LIN {X 0,Y 368.293,Z 314.692,A -85,B 0,C 180,E1 -12573.966,E2 -12573.966} C_VEL
LIN {X 0,Y 368.178,Z 320.417,A -85,B 0,C 180,E1 -12577.556,E2 -12577.556} C_VEL
LIN {X 0,Y 368.144,Z 324.235,A -85,B 0,C 180,E1 -12579.902,E2 -12579.902} C_VEL
LIN {X 0,Y 368.132,Z 327.336,A -85,B 0,C 180,E1 -12581.747,E2 -12581.747} C_VEL
LIN {X 0,Y 370.901,Z 341.005,A -85,B 0,C 180,E1 -12582.407,E2 -12582.407} C_VEL
LIN {X 0,Y 372.726,Z 351.323,A -85,B 0,C 180,E1 -12583.051,E2 -12583.051} C_VEL
LIN {X 0,Y 372.036,Z 364.185,A -85,B 0,C 180,E1 -12583.962,E2 -12583.962} C_VEL
LIN {X 0,Y 371.306,Z 375.959,A -85,B 0,C 180,E1 -12585.036,E2 -12585.036} C_VEL
LIN {X 0,Y 370.622,Z 386.995,A -85,B 0,C 180,E1 -12586.288,E2 -12586.288} C_VEL
LIN {X 0,Y 369.859,Z 396.767,A -85,B 0,C 180,E1 -12587.656,E2 -12587.656} C_VEL
LIN {X 0,Y 369.188,Z 406.325,A -85,B 0,C 180,E1 -12589.304,E2 -12589.304} C_VEL
LIN {X 0,Y 368.622,Z 413.953,A -85,B 0,C 180,E1 -12590.95,E2 -12590.95} C_VEL
LIN {X 0,Y 368.197,Z 420.432,A -85,B 0,C 180,E1 -12592.693,E2 -12592.693} C_VEL
LIN {X 0,Y 367.947,Z 425.635,A -85,B 0,C 180,E1 -12594.52,E2 -12594.52} C_VEL
LIN {X 0,Y 367.836,Z 428.082,A -85,B 0,C 180,E1 -12595.617,E2 -12595.617} C_VEL
LIN {X 0,Y 367.823,Z 430.069,A -85,B 0,C 180,E1 -12596.714,E2 -12596.714} C_VEL
LIN {X 0,Y 367.74,Z 431.56,A -85,B 0,C 180,E1 -12597.809,E2 -12597.809} C_VEL
LIN {X 0,Y 367.646,Z 432.642,A -85,B 0,C 180,E1 -12598.905,E2 -12598.905} C_VEL
LIN {X 0,Y 367.637,Z 433.299,A -85,B 0,C 180,E1 -12600,E2 -12600} C_VEL
LIN {X 0,Y 367.683,Z 433.487,A -85,B 0,C 180,E1 -12601.095,E2 -12601.095} C_VEL
LIN {X 0,Y 367.802,Z 433.269,A -85,B 0,C 180,E1 -12602.19,E2 -12602.19} C_VEL
LIN {X 0,Y 367.965,Z 432.627,A -85,B 0,C 180,E1 -12603.285,E2 -12603.285} C_VEL
LIN {X 0,Y 368.17,Z 431.513,A -85,B 0,C 180,E1 -12604.379,E2 -12604.379} C_VEL
LIN {X 0,Y 368.307,Z 429.993,A -85,B 0,C 180,E1 -12605.475,E2 -12605.475} C_VEL
LIN {X 0,Y 368.614,Z 426.762,A -85,B 0,C 180,E1 -12607.157,E2 -12607.157} C_VEL
LIN {X 0,Y 369.223,Z 422.567,A -85,B 0,C 180,E1 -12608.759,E2 -12608.759} C_VEL
LIN {X 0,Y 370.013,Z 415.974,A -85,B 0,C 180,E1 -12610.672,E2 -12610.672} C_VEL
LIN {X 0,Y 370.794,Z 408.79,A -85,B 0,C 180,E1 -12612.312,E2 -12612.312} C_VEL
LIN {X 0,Y 371.912,Z 399.78,A -85,B 0,C 180,E1 -12613.942,E2 -12613.942} C_VEL
LIN {X 0,Y 372.991,Z 390.605,A -85,B 0,C 180,E1 -12615.295,E2 -12615.295} C_VEL
LIN {X 0,Y 374.108,Z 379.922,A -85,B 0,C 180,E1 -12616.57,E2 -12616.57} C_VEL
LIN {X 0,Y 375.291,Z 367.919,A -85,B 0,C 180,E1 -12617.717,E2 -12617.717} C_VEL
LIN {X 0,Y 376.322,Z 355.559,A -85,B 0,C 180,E1 -12618.649,E2 -12618.649} C_VEL
LIN {X 0,Y 373.799,Z 345.042,A -85,B 0,C 180,E1 -12619.536,E2 -12619.536} C_VEL
LIN {X 0,Y 369.814,Z 333.869,A -85,B 0,C 180,E1 -12620.45,E2 -12620.45} C_VEL
LIN {X 0,Y 369.281,Z 332.067,A -85,B 0,C 180,E1 -12620.593,E2 -12620.593} C_VEL
LIN {X 0,Y 369.513,Z 325.412,A -85,B 0,C 180,E1 -12624.736,E2 -12624.736} C_VEL
LIN {X 0,Y 369.884,Z 318.305,A -85,B 0,C 180,E1 -12629.07,E2 -12629.07} C_VEL
LIN {X 0,Y 370.318,Z 312.164,A -85,B 0,C 180,E1 -12632.73,E2 -12632.73} C_VEL
LIN {X 0,Y 370.032,Z 308.99,A -85,B 0,C 180,E1 -12634.736,E2 -12634.736} C_VEL
LIN {X 0,Y 368.959,Z 303.753,A -85,B 0,C 180,E1 -12638.248,E2 -12638.248} C_VEL
LIN {X 0,Y 368.903,Z 303.535,A -85,B 0,C 180,E1 -12638.953,E2 -12638.953} C_VEL
LIN {X 0,Y 368.882,Z 303.536,A -85,B 0,C 180,E1 -12642.009,E2 -12642.009} C_VEL
LIN {X 0,Y 368.969,Z 303.673,A -85,B 0,C 180,E1 -12643.414,E2 -12643.414} C_VEL
LIN {X 0,Y 370.283,Z 310.676,A -85,B 0,C 180,E1 -12646.899,E2 -12646.899} C_VEL
LIN {X 0,Y 371.896,Z 318.9,A -85,B 0,C 180,E1 -12650.788,E2 -12650.788} C_VEL
LIN {X 0,Y 372.574,Z 323.529,A -85,B 0,C 180,E1 -12652.87,E2 -12652.87} C_VEL
LIN {X 0,Y 372.208,Z 328.239,A -85,B 0,C 180,E1 -12654.861,E2 -12654.861} C_VEL
LIN {X 0,Y 371.167,Z 337.939,A -85,B 0,C 180,E1 -12658.829,E2 -12658.829} C_VEL
LIN {X 0,Y 370.182,Z 348.156,A -85,B 0,C 180,E1 -12662.893,E2 -12662.893} C_VEL
LIN {X 0,Y 369.444,Z 357.311,A -85,B 0,C 180,E1 -12666.454,E2 -12666.454} C_VEL
LIN {X 0,Y 368.798,Z 366.881,A -85,B 0,C 180,E1 -12670.121,E2 -12670.121} C_VEL
LIN {X 0,Y 370.827,Z 380.273,A -85,B 0,C 180,E1 -12670.828,E2 -12670.828} C_VEL
LIN {X 0,Y 372.37,Z 395.112,A -85,B 0,C 180,E1 -12671.806,E2 -12671.806} C_VEL
LIN {X 0,Y 373.203,Z 403.232,A -85,B 0,C 180,E1 -12672.464,E2 -12672.464} C_VEL
LIN {X 0,Y 372.141,Z 415.707,A -85,B 0,C 180,E1 -12673.544,E2 -12673.544} C_VEL
LIN {X 0,Y 371.014,Z 427.836,A -85,B 0,C 180,E1 -12674.838,E2 -12674.838} C_VEL
LIN {X 0,Y 370.307,Z 436.542,A -85,B 0,C 180,E1 -12675.996,E2 -12675.996} C_VEL
LIN {X 0,Y 369.48,Z 445.02,A -85,B 0,C 180,E1 -12677.365,E2 -12677.365} C_VEL
LIN {X 0,Y 368.646,Z 453.276,A -85,B 0,C 180,E1 -12679.01,E2 -12679.01} C_VEL
LIN {X 0,Y 368.16,Z 459.921,A -85,B 0,C 180,E1 -12680.662,E2 -12680.662} C_VEL
LIN {X 0,Y 367.808,Z 465.21,A -85,B 0,C 180,E1 -12682.313,E2 -12682.313} C_VEL
LIN {X 0,Y 367.693,Z 468.753,A -85,B 0,C 180,E1 -12683.679,E2 -12683.679} C_VEL
LIN {X 0,Y 367.561,Z 472.55,A -85,B 0,C 180,E1 -12685.614,E2 -12685.614} C_VEL
LIN {X 0,Y 367.561,Z 474.042,A -85,B 0,C 180,E1 -12686.712,E2 -12686.712} C_VEL
LIN {X 0,Y 367.596,Z 475.113,A -85,B 0,C 180,E1 -12687.809,E2 -12687.809} C_VEL
LIN {X 0,Y 367.68,Z 475.776,A -85,B 0,C 180,E1 -12688.905,E2 -12688.905} C_VEL
LIN {X 0,Y 367.674,Z 475.968,A -85,B 0,C 180,E1 -12690,E2 -12690} C_VEL
LIN {X 0,Y 367.674,Z 475.73,A -85,B 0,C 180,E1 -12691.095,E2 -12691.095} C_VEL
LIN {X 0,Y 367.623,Z 475.08,A -85,B 0,C 180,E1 -12692.191,E2 -12692.191} C_VEL
LIN {X 0,Y 367.547,Z 473.974,A -85,B 0,C 180,E1 -12693.289,E2 -12693.289} C_VEL
LIN {X 0,Y 367.571,Z 472.414,A -85,B 0,C 180,E1 -12694.386,E2 -12694.386} C_VEL
LIN {X 0,Y 367.732,Z 468.044,A -85,B 0,C 180,E1 -12696.585,E2 -12696.585} C_VEL
LIN {X 0,Y 367.909,Z 463.575,A -85,B 0,C 180,E1 -12698.237,E2 -12698.237} C_VEL
LIN {X 0,Y 368.322,Z 457.886,A -85,B 0,C 180,E1 -12699.888,E2 -12699.888} C_VEL
LIN {X 0,Y 368.894,Z 450.724,A -85,B 0,C 180,E1 -12701.539,E2 -12701.539} C_VEL
LIN {X 0,Y 369.76,Z 441.784,A -85,B 0,C 180,E1 -12703.184,E2 -12703.184} C_VEL
LIN {X 0,Y 370.829,Z 430.162,A -85,B 0,C 180,E1 -12704.931,E2 -12704.931} C_VEL
LIN {X 0,Y 372.024,Z 418.794,A -85,B 0,C 180,E1 -12706.32,E2 -12706.32} C_VEL
LIN {X 0,Y 373.408,Z 406.425,A -85,B 0,C 180,E1 -12707.526,E2 -12707.526} C_VEL
LIN {X 0,Y 373.418,Z 401.589,A -85,B 0,C 180,E1 -12707.95,E2 -12707.95} C_VEL
LIN {X 0,Y 372.561,Z 389.175,A -85,B 0,C 180,E1 -12708.946,E2 -12708.946} C_VEL
LIN {X 0,Y 371.454,Z 377.338,A -85,B 0,C 180,E1 -12709.731,E2 -12709.731} C_VEL
LIN {X 0,Y 369.366,Z 365.834,A -85,B 0,C 180,E1 -12710.417,E2 -12710.417} C_VEL
LIN {X 0,Y 368.722,Z 362.563,A -85,B 0,C 180,E1 -12710.631,E2 -12710.631} C_VEL
LIN {X 0,Y 369.355,Z 353.705,A -85,B 0,C 180,E1 -12714.03,E2 -12714.03} C_VEL
LIN {X 0,Y 370.072,Z 344.511,A -85,B 0,C 180,E1 -12717.728,E2 -12717.728} C_VEL
LIN {X 0,Y 371.079,Z 335.65,A -85,B 0,C 180,E1 -12721.54,E2 -12721.54} C_VEL
LIN {X 0,Y 372.163,Z 328.029,A -85,B 0,C 180,E1 -12725.138,E2 -12725.138} C_VEL
LIN {X 0,Y 372.658,Z 324.25,A -85,B 0,C 180,E1 -12727.121,E2 -12727.121} C_VEL
LIN {X 0,Y 372.228,Z 320.752,A -85,B 0,C 180,E1 -12729.275,E2 -12729.275} C_VEL
LIN {X 0,Y 371.416,Z 316.482,A -85,B 0,C 180,E1 -12732.441,E2 -12732.441} C_VEL
LIN {X 0,Y 370.833,Z 313.284,A -85,B 0,C 180,E1 -12735.475,E2 -12735.475} C_VEL
LIN {X 0,Y 370.417,Z 311.076,A -85,B 0,C 180,E1 -12738.389,E2 -12738.389} C_VEL
LIN {X 0,Y 370.16,Z 309.682,A -85,B 0,C 180,E1 -12741.204,E2 -12741.204} C_VEL
LIN {X 0,Y 369.927,Z 308.905,A -85,B 0,C 180,E1 -12744.779,E2 -12744.779} C_VEL
LIN {X 0,Y 369.886,Z 308.938,A -85,B 0,C 180,E1 -12747.858,E2 -12747.858} C_VEL
LIN {X 0,Y 370.009,Z 309.705,A -85,B 0,C 180,E1 -12751.65,E2 -12751.65} C_VEL
LIN {X 0,Y 370.086,Z 310.561,A -85,B 0,C 180,E1 -12754.102,E2 -12754.102} C_VEL
LIN {X 0,Y 370.024,Z 311.641,A -85,B 0,C 180,E1 -12756.493,E2 -12756.493} C_VEL
LIN {X 0,Y 369.869,Z 313.391,A -85,B 0,C 180,E1 -12759.546,E2 -12759.546} C_VEL
LIN {X 0,Y 375.177,Z 326.38,A -85,B 0,C 180,E1 -12760.749,E2 -12760.749} C_VEL
LIN {X 0,Y 377.211,Z 332.806,A -85,B 0,C 180,E1 -12761.355,E2 -12761.355} C_VEL
LIN {X 0,Y 376.25,Z 345.093,A -85,B 0,C 180,E1 -12762.295,E2 -12762.295} C_VEL
LIN {X 0,Y 375.212,Z 355.755,A -85,B 0,C 180,E1 -12763.317,E2 -12763.317} C_VEL
LIN {X 0,Y 374.169,Z 365.672,A -85,B 0,C 180,E1 -12764.475,E2 -12764.475} C_VEL
LIN {X 0,Y 373.088,Z 375.04,A -85,B 0,C 180,E1 -12765.825,E2 -12765.825} C_VEL
LIN {X 0,Y 371.984,Z 384.167,A -85,B 0,C 180,E1 -12767.451,E2 -12767.451} C_VEL
LIN {X 0,Y 370.925,Z 391.487,A -85,B 0,C 180,E1 -12769.078,E2 -12769.078} C_VEL
LIN {X 0,Y 370.181,Z 397.689,A -85,B 0,C 180,E1 -12770.838,E2 -12770.838} C_VEL
LIN {X 0,Y 369.461,Z 401.878,A -85,B 0,C 180,E1 -12772.348,E2 -12772.348} C_VEL
LIN {X 0,Y 369.123,Z 404.297,A -85,B 0,C 180,E1 -12773.44,E2 -12773.44} C_VEL
LIN {X 0,Y 368.943,Z 406.185,A -85,B 0,C 180,E1 -12774.535,E2 -12774.535} C_VEL
LIN {X 0,Y 368.636,Z 407.667,A -85,B 0,C 180,E1 -12775.626,E2 -12775.626} C_VEL
LIN {X 0,Y 368.304,Z 408.741,A -85,B 0,C 180,E1 -12776.718,E2 -12776.718} C_VEL
LIN {X 0,Y 368.069,Z 409.353,A -85,B 0,C 180,E1 -12777.811,E2 -12777.811} C_VEL
LIN {X 0,Y 367.947,Z 409.528,A -85,B 0,C 180,E1 -12778.906,E2 -12778.906} C_VEL
LIN {X 0,Y 367.9,Z 409.292,A -85,B 0,C 180,E1 -12780,E2 -12780} C_VEL
LIN {X 0,Y 367.924,Z 408.635,A -85,B 0,C 180,E1 -12781.095,E2 -12781.095} C_VEL
LIN {X 0,Y 368.046,Z 407.513,A -85,B 0,C 180,E1 -12782.189,E2 -12782.189} C_VEL
LIN {X 0,Y 368.166,Z 405.984,A -85,B 0,C 180,E1 -12783.283,E2 -12783.283} C_VEL
LIN {X 0,Y 368.432,Z 402.847,A -85,B 0,C 180,E1 -12784.924,E2 -12784.924} C_VEL
LIN {X 0,Y 368.507,Z 398.641,A -85,B 0,C 180,E1 -12786.571,E2 -12786.571} C_VEL
LIN {X 0,Y 368.886,Z 393.227,A -85,B 0,C 180,E1 -12788.215,E2 -12788.215} C_VEL
LIN {X 0,Y 369.311,Z 386.432,A -85,B 0,C 180,E1 -12789.862,E2 -12789.862} C_VEL
LIN {X 0,Y 369.939,Z 377.981,A -85,B 0,C 180,E1 -12791.506,E2 -12791.506} C_VEL
LIN {X 0,Y 370.554,Z 369.405,A -85,B 0,C 180,E1 -12792.877,E2 -12792.877} C_VEL
LIN {X 0,Y 371.324,Z 358.953,A -85,B 0,C 180,E1 -12794.244,E2 -12794.244} C_VEL
LIN {X 0,Y 372.069,Z 346.412,A -85,B 0,C 180,E1 -12795.562,E2 -12795.562} C_VEL
LIN {X 0,Y 372.687,Z 334.118,A -85,B 0,C 180,E1 -12796.572,E2 -12796.572} C_VEL
LIN {X 0,Y 373.108,Z 324.805,A -85,B 0,C 180,E1 -12797.187,E2 -12797.187} C_VEL
LIN {X 0,Y 369.814,Z 310.534,A -85,B 0,C 180,E1 -12798.046,E2 -12798.046} C_VEL
LIN {X 0,Y 368.184,Z 303.626,A -85,B 0,C 180,E1 -12798.395,E2 -12798.395} C_VEL
LIN {X 0,Y 368.516,Z 303.575,A -85,B 0,C 180,E1 -12801.245,E2 -12801.245} C_VEL
LIN {X 0,Y 368.767,Z 303.553,A -85,B 0,C 180,E1 -12803.824,E2 -12803.824} C_VEL
LIN {X 0,Y 368.916,Z 303.525,A -85,B 0,C 180,E1 -12806.443,E2 -12806.443} C_VEL
LIN {X 0,Y 368.916,Z 303.529,A -85,B 0,C 180,E1 -12809.69,E2 -12809.69} C_VEL
LIN {X 0,Y 368.901,Z 303.533,A -85,B 0,C 180,E1 -12813.044,E2 -12813.044} C_VEL
LIN {X 0,Y 368.92,Z 303.53,A -85,B 0,C 180,E1 -12816.197,E2 -12816.197} C_VEL
LIN {X 0,Y 368.905,Z 303.531,A -85,B 0,C 180,E1 -12818.953,E2 -12818.953} C_VEL
LIN {X 0,Y 368.884,Z 303.537,A -85,B 0,C 180,E1 -12822.009,E2 -12822.009} C_VEL
LIN {X 0,Y 368.883,Z 303.534,A -85,B 0,C 180,E1 -12825.176,E2 -12825.176} C_VEL
LIN {X 0,Y 368.885,Z 303.535,A -85,B 0,C 180,E1 -12828.178,E2 -12828.178} C_VEL
LIN {X 0,Y 368.91,Z 303.534,A -85,B 0,C 180,E1 -12831.36,E2 -12831.36} C_VEL
LIN {X 0,Y 368.881,Z 303.539,A -85,B 0,C 180,E1 -12833.799,E2 -12833.799} C_VEL
LIN {X 0,Y 368.808,Z 303.601,A -85,B 0,C 180,E1 -12835.96,E2 -12835.96} C_VEL
LIN {X 0,Y 368.572,Z 308.503,A -85,B 0,C 180,E1 -12839.101,E2 -12839.101} C_VEL
LIN {X 0,Y 368.516,Z 312.27,A -85,B 0,C 180,E1 -12841.525,E2 -12841.525} C_VEL
LIN {X 0,Y 368.382,Z 318.111,A -85,B 0,C 180,E1 -12845.183,E2 -12845.183} C_VEL
LIN {X 0,Y 368.376,Z 324.094,A -85,B 0,C 180,E1 -12848.747,E2 -12848.747} C_VEL
LIN {X 0,Y 368.374,Z 327.317,A -85,B 0,C 180,E1 -12850.443,E2 -12850.443} C_VEL
LIN {X 0,Y 371.93,Z 340.357,A -85,B 0,C 180,E1 -12851.087,E2 -12851.087} C_VEL
LIN {X 0,Y 374.511,Z 351.672,A -85,B 0,C 180,E1 -12851.81,E2 -12851.81} C_VEL
LIN {X 0,Y 374.813,Z 355.874,A -85,B 0,C 180,E1 -12852.094,E2 -12852.094} C_VEL
LIN {X 0,Y 373.988,Z 367.324,A -85,B 0,C 180,E1 -12852.925,E2 -12852.925} C_VEL
LIN {X 0,Y 373.044,Z 378.613,A -85,B 0,C 180,E1 -12853.989,E2 -12853.989} C_VEL
LIN {X 0,Y 372.202,Z 389.01,A -85,B 0,C 180,E1 -12855.232,E2 -12855.232} C_VEL
LIN {X 0,Y 371.226,Z 398.28,A -85,B 0,C 180,E1 -12856.59,E2 -12856.59} C_VEL
LIN {X 0,Y 370.223,Z 407.2,A -85,B 0,C 180,E1 -12858.225,E2 -12858.225} C_VEL
LIN {X 0,Y 369.426,Z 414.361,A -85,B 0,C 180,E1 -12859.865,E2 -12859.865} C_VEL
LIN {X 0,Y 368.72,Z 420.921,A -85,B 0,C 180,E1 -12861.781,E2 -12861.781} C_VEL
LIN {X 0,Y 368.33,Z 425.227,A -85,B 0,C 180,E1 -12863.426,E2 -12863.426} C_VEL
LIN {X 0,Y 368.005,Z 427.501,A -85,B 0,C 180,E1 -12864.521,E2 -12864.521} C_VEL
LIN {X 0,Y 367.926,Z 429.344,A -85,B 0,C 180,E1 -12865.618,E2 -12865.618} C_VEL
LIN {X 0,Y 367.907,Z 430.748,A -85,B 0,C 180,E1 -12866.715,E2 -12866.715} C_VEL
LIN {X 0,Y 367.628,Z 432.356,A -85,B 0,C 180,E1 -12868.905,E2 -12868.905} C_VEL
LIN {X 0,Y 367.604,Z 432.59,A -85,B 0,C 180,E1 -12870,E2 -12870} C_VEL
LIN {X 0,Y 367.742,Z 431.812,A -85,B 0,C 180,E1 -12872.191,E2 -12872.191} C_VEL
LIN {X 0,Y 367.882,Z 430.847,A -85,B 0,C 180,E1 -12873.286,E2 -12873.286} C_VEL
LIN {X 0,Y 367.899,Z 429.498,A -85,B 0,C 180,E1 -12874.382,E2 -12874.382} C_VEL
LIN {X 0,Y 368.14,Z 426.646,A -85,B 0,C 180,E1 -12876.027,E2 -12876.027} C_VEL
LIN {X 0,Y 368.536,Z 422.768,A -85,B 0,C 180,E1 -12877.671,E2 -12877.671} C_VEL
LIN {X 0,Y 369.03,Z 417.746,A -85,B 0,C 180,E1 -12879.316,E2 -12879.316} C_VEL
LIN {X 0,Y 369.809,Z 411.399,A -85,B 0,C 180,E1 -12880.955,E2 -12880.955} C_VEL
LIN {X 0,Y 370.665,Z 403.513,A -85,B 0,C 180,E1 -12882.594,E2 -12882.594} C_VEL
LIN {X 0,Y 371.569,Z 395.448,A -85,B 0,C 180,E1 -12883.955,E2 -12883.955} C_VEL
LIN {X 0,Y 372.57,Z 385.545,A -85,B 0,C 180,E1 -12885.313,E2 -12885.313} C_VEL
LIN {X 0,Y 373.313,Z 375.766,A -85,B 0,C 180,E1 -12886.403,E2 -12886.403} C_VEL
LIN {X 0,Y 374.204,Z 365.147,A -85,B 0,C 180,E1 -12887.347,E2 -12887.347} C_VEL
LIN {X 0,Y 374.88,Z 353.869,A -85,B 0,C 180,E1 -12888.136,E2 -12888.136} C_VEL
LIN {X 0,Y 372.278,Z 341.681,A -85,B 0,C 180,E1 -12888.939,E2 -12888.939} C_VEL
LIN {X 0,Y 368.878,Z 329.095,A -85,B 0,C 180,E1 -12889.582,E2 -12889.582} C_VEL
LIN {X 0,Y 368.37,Z 327.121,A -85,B 0,C 180,E1 -12889.666,E2 -12889.666} C_VEL
LIN {X 0,Y 368.391,Z 321.258,A -85,B 0,C 180,E1 -12893.022,E2 -12893.022} C_VEL
LIN {X 0,Y 368.379,Z 320.193,A -85,B 0,C 180,E1 -12893.66,E2 -12893.66} C_VEL
LIN {X 0,Y 367.704,Z 318.867,A -85,B 0,C 180,E1 -12894.55,E2 -12894.55} C_VEL
LIN {X 0,Y 364.873,Z 316.949,A -85,B 0,C 180,E1 -12896.006,E2 -12896.006} C_VEL
LIN {X 0,Y 362.504,Z 315.428,A -85,B 0,C 180,E1 -12897.184,E2 -12897.184} C_VEL
LIN {X 0,Y 361.511,Z 314.156,A -85,B 0,C 180,E1 -12898.09,E2 -12898.09} C_VEL
LIN {X 0,Y 361.442,Z 313.674,A -85,B 0,C 180,E1 -12898.395,E2 -12898.395} C_VEL
LIN {X 0,Y 361.596,Z 308.64,A -85,B 0,C 180,E1 -12901.653,E2 -12901.653} C_VEL
LIN {X 0,Y 361.789,Z 304.422,A -85,B 0,C 180,E1 -12904.372,E2 -12904.372} C_VEL
LIN {X 0,Y 361.854,Z 304.414,A -85,B 0,C 180,E1 -12907.221,E2 -12907.221} C_VEL
LIN {X 0,Y 361.838,Z 304.416,A -85,B 0,C 180,E1 -12910.755,E2 -12910.755} C_VEL
LIN {X 0,Y 361.819,Z 304.418,A -85,B 0,C 180,E1 -12914.368,E2 -12914.368} C_VEL
LIN {X 0,Y 361.838,Z 304.416,A -85,B 0,C 180,E1 -12917.568,E2 -12917.568} C_VEL
LIN {X 0,Y 361.872,Z 304.409,A -85,B 0,C 180,E1 -12920.973,E2 -12920.973} C_VEL
LIN {X 0,Y 361.765,Z 304.421,A -85,B 0,C 180,E1 -12924.351,E2 -12924.351} C_VEL
LIN {X 0,Y 361.584,Z 304.489,A -85,B 0,C 180,E1 -12927.028,E2 -12927.028} C_VEL
LIN {X 0,Y 361.278,Z 310.934,A -85,B 0,C 180,E1 -12931.092,E2 -12931.092} C_VEL
LIN {X 0,Y 361.19,Z 316.609,A -85,B 0,C 180,E1 -12934.654,E2 -12934.654} C_VEL
LIN {X 0,Y 361.122,Z 320.505,A -85,B 0,C 180,E1 -12937.093,E2 -12937.093} C_VEL
LIN {X 0,Y 361.05,Z 326.236,A -85,B 0,C 180,E1 -12940.676,E2 -12940.676} C_VEL
LIN {X 0,Y 361.045,Z 327.547,A -85,B 0,C 180,E1 -12941.488,E2 -12941.488} C_VEL
LIN {X 0,Y 363.676,Z 340.651,A -85,B 0,C 180,E1 -12942.13,E2 -12942.13} C_VEL
LIN {X 0,Y 365.641,Z 350.928,A -85,B 0,C 180,E1 -12942.782,E2 -12942.782} C_VEL
LIN {X 0,Y 365.149,Z 363.106,A -85,B 0,C 180,E1 -12943.651,E2 -12943.651} C_VEL
LIN {X 0,Y 364.384,Z 375.234,A -85,B 0,C 180,E1 -12944.745,E2 -12944.745} C_VEL
LIN {X 0,Y 363.704,Z 386.455,A -85,B 0,C 180,E1 -12946.022,E2 -12946.022} C_VEL
LIN {X 0,Y 362.867,Z 396.447,A -85,B 0,C 180,E1 -12947.415,E2 -12947.415} C_VEL
LIN {X 0,Y 362.174,Z 406.145,A -85,B 0,C 180,E1 -12949.094,E2 -12949.094} C_VEL
LIN {X 0,Y 361.587,Z 413.912,A -85,B 0,C 180,E1 -12950.773,E2 -12950.773} C_VEL
LIN {X 0,Y 361.136,Z 420.244,A -85,B 0,C 180,E1 -12952.48,E2 -12952.48} C_VEL
LIN {X 0,Y 360.872,Z 425.806,A -85,B 0,C 180,E1 -12954.412,E2 -12954.412} C_VEL
LIN {X 0,Y 360.727,Z 429.373,A -85,B 0,C 180,E1 -12956.09,E2 -12956.09} C_VEL
LIN {X 0,Y 360.662,Z 431.891,A -85,B 0,C 180,E1 -12957.766,E2 -12957.766} C_VEL
LIN {X 0,Y 360.581,Z 433.016,A -85,B 0,C 180,E1 -12958.883,E2 -12958.883} C_VEL
LIN {X 0,Y 360.568,Z 433.732,A -85,B 0,C 180,E1 -12960,E2 -12960} C_VEL
LIN {X 0,Y 360.616,Z 433.971,A -85,B 0,C 180,E1 -12961.117,E2 -12961.117} C_VEL
LIN {X 0,Y 360.742,Z 433.788,A -85,B 0,C 180,E1 -12962.233,E2 -12962.233} C_VEL
LIN {X 0,Y 360.917,Z 433.197,A -85,B 0,C 180,E1 -12963.349,E2 -12963.349} C_VEL
LIN {X 0,Y 361.133,Z 432.137,A -85,B 0,C 180,E1 -12964.465,E2 -12964.465} C_VEL
LIN {X 0,Y 361.267,Z 430.664,A -85,B 0,C 180,E1 -12965.582,E2 -12965.582} C_VEL
LIN {X 0,Y 361.587,Z 427.659,A -85,B 0,C 180,E1 -12967.227,E2 -12967.227} C_VEL
LIN {X 0,Y 362.276,Z 423.387,A -85,B 0,C 180,E1 -12968.928,E2 -12968.928} C_VEL
LIN {X 0,Y 363.1,Z 416.909,A -85,B 0,C 180,E1 -12970.878,E2 -12970.878} C_VEL
LIN {X 0,Y 363.955,Z 409.875,A -85,B 0,C 180,E1 -12972.547,E2 -12972.547} C_VEL
LIN {X 0,Y 365.132,Z 401.023,A -85,B 0,C 180,E1 -12974.206,E2 -12974.206} C_VEL
LIN {X 0,Y 366.272,Z 391.97,A -85,B 0,C 180,E1 -12975.583,E2 -12975.583} C_VEL
LIN {X 0,Y 367.425,Z 382.046,A -85,B 0,C 180,E1 -12976.831,E2 -12976.831} C_VEL
LIN {X 0,Y 368.716,Z 370.023,A -85,B 0,C 180,E1 -12978.043,E2 -12978.043} C_VEL
LIN {X 0,Y 369.806,Z 358.016,A -85,B 0,C 180,E1 -12978.993,E2 -12978.993} C_VEL
LIN {X 0,Y 369.115,Z 353.419,A -85,B 0,C 180,E1 -12979.391,E2 -12979.391} C_VEL
LIN {X 0,Y 366.4,Z 343.698,A -85,B 0,C 180,E1 -12980.262,E2 -12980.262} C_VEL
LIN {X 0,Y 362.394,Z 332.714,A -85,B 0,C 180,E1 -12981.228,E2 -12981.228} C_VEL
LIN {X 0,Y 362.625,Z 327.765,A -85,B 0,C 180,E1 -12984.369,E2 -12984.369} C_VEL
LIN {X 0,Y 362.839,Z 322.439,A -85,B 0,C 180,E1 -12987.702,E2 -12987.702} C_VEL
LIN {X 0,Y 363.251,Z 317.385,A -85,B 0,C 180,E1 -12990.844,E2 -12990.844} C_VEL
LIN {X 0,Y 363.547,Z 314.265,A -85,B 0,C 180,E1 -12992.771,E2 -12992.771} C_VEL
LIN {X 0,Y 363.302,Z 311.172,A -85,B 0,C 180,E1 -12994.797,E2 -12994.797} C_VEL
LIN {X 0,Y 362.316,Z 306.185,A -85,B 0,C 180,E1 -12998.369,E2 -12998.369} C_VEL
LIN {X 0,Y 361.856,Z 304.412,A -85,B 0,C 180,E1 -12999.861,E2 -12999.861} C_VEL
LIN {X 0,Y 361.87,Z 304.485,A -85,B 0,C 180,E1 -13003.014,E2 -13003.014} C_VEL
LIN {X 0,Y 363.2,Z 311.378,A -85,B 0,C 180,E1 -13006.521,E2 -13006.521} C_VEL
LIN {X 0,Y 364.815,Z 319.672,A -85,B 0,C 180,E1 -13010.526,E2 -13010.526} C_VEL
LIN {X 0,Y 365.559,Z 324.507,A -85,B 0,C 180,E1 -13012.746,E2 -13012.746} C_VEL
LIN {X 0,Y 365.209,Z 329.13,A -85,B 0,C 180,E1 -13014.738,E2 -13014.738} C_VEL
LIN {X 0,Y 364.172,Z 338.366,A -85,B 0,C 180,E1 -13018.596,E2 -13018.596} C_VEL
LIN {X 0,Y 363.224,Z 347.547,A -85,B 0,C 180,E1 -13022.33,E2 -13022.33} C_VEL
LIN {X 0,Y 362.471,Z 356.694,A -85,B 0,C 180,E1 -13025.973,E2 -13025.973} C_VEL
LIN {X 0,Y 361.804,Z 365.665,A -85,B 0,C 180,E1 -13029.485,E2 -13029.485} C_VEL
LIN {X 0,Y 363.812,Z 376.83,A -85,B 0,C 180,E1 -13030.131,E2 -13030.131} C_VEL
LIN {X 0,Y 365.264,Z 390.15,A -85,B 0,C 180,E1 -13030.993,E2 -13030.993} C_VEL
LIN {X 0,Y 366.39,Z 403.054,A -85,B 0,C 180,E1 -13032.033,E2 -13032.033} C_VEL
LIN {X 0,Y 366.14,Z 409.03,A -85,B 0,C 180,E1 -13032.547,E2 -13032.547} C_VEL
LIN {X 0,Y 364.965,Z 420.178,A -85,B 0,C 180,E1 -13033.643,E2 -13033.643} C_VEL
LIN {X 0,Y 363.786,Z 431.272,A -85,B 0,C 180,E1 -13035.006,E2 -13035.006} C_VEL
LIN {X 0,Y 362.979,Z 439.782,A -85,B 0,C 180,E1 -13036.279,E2 -13036.279} C_VEL
LIN {X 0,Y 362.058,Z 448.962,A -85,B 0,C 180,E1 -13037.955,E2 -13037.955} C_VEL
LIN {X 0,Y 361.385,Z 456.412,A -85,B 0,C 180,E1 -13039.637,E2 -13039.637} C_VEL
LIN {X 0,Y 360.979,Z 461.51,A -85,B 0,C 180,E1 -13041.039,E2 -13041.039} C_VEL
LIN {X 0,Y 360.696,Z 466.454,A -85,B 0,C 180,E1 -13042.724,E2 -13042.724} C_VEL
LIN {X 0,Y 360.573,Z 470.26,A -85,B 0,C 180,E1 -13044.407,E2 -13044.407} C_VEL
LIN {X 0,Y 360.496,Z 472.218,A -85,B 0,C 180,E1 -13045.527,E2 -13045.527} C_VEL
LIN {X 0,Y 360.469,Z 473.688,A -85,B 0,C 180,E1 -13046.647,E2 -13046.647} C_VEL
LIN {X 0,Y 360.498,Z 474.745,A -85,B 0,C 180,E1 -13047.765,E2 -13047.765} C_VEL
LIN {X 0,Y 360.608,Z 475.391,A -85,B 0,C 180,E1 -13048.883,E2 -13048.883} C_VEL
LIN {X 0,Y 360.603,Z 475.558,A -85,B 0,C 180,E1 -13050,E2 -13050} C_VEL
LIN {X 0,Y 360.603,Z 475.307,A -85,B 0,C 180,E1 -13051.117,E2 -13051.117} C_VEL
LIN {X 0,Y 360.526,Z 474.639,A -85,B 0,C 180,E1 -13052.234,E2 -13052.234} C_VEL
LIN {X 0,Y 360.457,Z 473.498,A -85,B 0,C 180,E1 -13053.353,E2 -13053.353} C_VEL
LIN {X 0,Y 360.558,Z 469.979,A -85,B 0,C 180,E1 -13055.593,E2 -13055.593} C_VEL
LIN {X 0,Y 360.689,Z 466.257,A -85,B 0,C 180,E1 -13057.276,E2 -13057.276} C_VEL
LIN {X 0,Y 360.981,Z 461.391,A -85,B 0,C 180,E1 -13058.961,E2 -13058.961} C_VEL
LIN {X 0,Y 361.441,Z 455.237,A -85,B 0,C 180,E1 -13060.645,E2 -13060.645} C_VEL
LIN {X 0,Y 362.192,Z 447.572,A -85,B 0,C 180,E1 -13062.324,E2 -13062.324} C_VEL
LIN {X 0,Y 363.4,Z 436.31,A -85,B 0,C 180,E1 -13064.275,E2 -13064.275} C_VEL
LIN {X 0,Y 364.329,Z 426.725,A -85,B 0,C 180,E1 -13065.668,E2 -13065.668} C_VEL
LIN {X 0,Y 365.706,Z 415.158,A -85,B 0,C 180,E1 -13067.042,E2 -13067.042} C_VEL
LIN {X 0,Y 366.769,Z 405.302,A -85,B 0,C 180,E1 -13067.998,E2 -13067.998} C_VEL
LIN {X 0,Y 366.015,Z 391.747,A -85,B 0,C 180,E1 -13069.185,E2 -13069.185} C_VEL
LIN {X 0,Y 365.172,Z 380.398,A -85,B 0,C 180,E1 -13070.008,E2 -13070.008} C_VEL
LIN {X 0,Y 363.194,Z 368.413,A -85,B 0,C 180,E1 -13070.8,E2 -13070.8} C_VEL
LIN {X 0,Y 361.742,Z 361.708,A -85,B 0,C 180,E1 -13071.221,E2 -13071.221} C_VEL
LIN {X 0,Y 362.421,Z 352.94,A -85,B 0,C 180,E1 -13074.695,E2 -13074.695} C_VEL
LIN {X 0,Y 363.176,Z 344.295,A -85,B 0,C 180,E1 -13078.302,E2 -13078.302} C_VEL
LIN {X 0,Y 364.171,Z 336.261,A -85,B 0,C 180,E1 -13081.882,E2 -13081.882} C_VEL
LIN {X 0,Y 365.25,Z 329.334,A -85,B 0,C 180,E1 -13085.257,E2 -13085.257} C_VEL
LIN {X 0,Y 365.758,Z 325.665,A -85,B 0,C 180,E1 -13087.248,E2 -13087.248} C_VEL
LIN {X 0,Y 365.276,Z 321.882,A -85,B 0,C 180,E1 -13089.681,E2 -13089.681} C_VEL
LIN {X 0,Y 364.49,Z 317.773,A -85,B 0,C 180,E1 -13092.886,E2 -13092.886} C_VEL
LIN {X 0,Y 363.915,Z 314.754,A -85,B 0,C 180,E1 -13095.954,E2 -13095.954} C_VEL
LIN {X 0,Y 363.509,Z 312.636,A -85,B 0,C 180,E1 -13098.94,E2 -13098.94} C_VEL
LIN {X 0,Y 363.245,Z 311.374,A -85,B 0,C 180,E1 -13101.747,E2 -13101.747} C_VEL
LIN {X 0,Y 363.065,Z 310.75,A -85,B 0,C 180,E1 -13104.499,E2 -13104.499} C_VEL
LIN {X 0,Y 363.004,Z 310.636,A -85,B 0,C 180,E1 -13107.173,E2 -13107.173} C_VEL
LIN {X 0,Y 363.051,Z 311.1,A -85,B 0,C 180,E1 -13110.589,E2 -13110.589} C_VEL
LIN {X 0,Y 363.143,Z 311.968,A -85,B 0,C 180,E1 -13113.569,E2 -13113.569} C_VEL
LIN {X 0,Y 363.115,Z 312.964,A -85,B 0,C 180,E1 -13116.018,E2 -13116.018} C_VEL
LIN {X 0,Y 362.949,Z 314.51,A -85,B 0,C 180,E1 -13118.916,E2 -13118.916} C_VEL
LIN {X 0,Y 364.207,Z 317.424,A -85,B 0,C 180,E1 -13119.198,E2 -13119.198} C_VEL
LIN {X 0,Y 368.972,Z 328.857,A -85,B 0,C 180,E1 -13120.349,E2 -13120.349} C_VEL
LIN {X 0,Y 370.798,Z 334.476,A -85,B 0,C 180,E1 -13120.927,E2 -13120.927} C_VEL
LIN {X 0,Y 369.716,Z 347.873,A -85,B 0,C 180,E1 -13122.007,E2 -13122.007} C_VEL
LIN {X 0,Y 368.527,Z 359.123,A -85,B 0,C 180,E1 -13123.156,E2 -13123.156} C_VEL
LIN {X 0,Y 367.321,Z 369.399,A -85,B 0,C 180,E1 -13124.463,E2 -13124.463} C_VEL
LIN {X 0,Y 366.145,Z 378.273,A -85,B 0,C 180,E1 -13125.834,E2 -13125.834} C_VEL
LIN {X 0,Y 365.022,Z 386.87,A -85,B 0,C 180,E1 -13127.49,E2 -13127.49} C_VEL
LIN {X 0,Y 363.968,Z 393.801,A -85,B 0,C 180,E1 -13129.148,E2 -13129.148} C_VEL
LIN {X 0,Y 363.302,Z 398.648,A -85,B 0,C 180,E1 -13130.606,E2 -13130.606} C_VEL
LIN {X 0,Y 362.525,Z 402.937,A -85,B 0,C 180,E1 -13132.201,E2 -13132.201} C_VEL
LIN {X 0,Y 362.165,Z 405.3,A -85,B 0,C 180,E1 -13133.314,E2 -13133.314} C_VEL
LIN {X 0,Y 361.938,Z 407.138,A -85,B 0,C 180,E1 -13134.428,E2 -13134.428} C_VEL
LIN {X 0,Y 361.619,Z 408.57,A -85,B 0,C 180,E1 -13135.541,E2 -13135.541} C_VEL
LIN {X 0,Y 361.275,Z 409.587,A -85,B 0,C 180,E1 -13136.654,E2 -13136.654} C_VEL
LIN {X 0,Y 361.028,Z 410.131,A -85,B 0,C 180,E1 -13137.769,E2 -13137.769} C_VEL
LIN {X 0,Y 360.898,Z 410.262,A -85,B 0,C 180,E1 -13138.884,E2 -13138.884} C_VEL
LIN {X 0,Y 360.848,Z 409.987,A -85,B 0,C 180,E1 -13140,E2 -13140} C_VEL
LIN {X 0,Y 360.876,Z 409.259,A -85,B 0,C 180,E1 -13141.116,E2 -13141.116} C_VEL
LIN {X 0,Y 360.986,Z 408.093,A -85,B 0,C 180,E1 -13142.232,E2 -13142.232} C_VEL
LIN {X 0,Y 361.19,Z 405.546,A -85,B 0,C 180,E1 -13143.905,E2 -13143.905} C_VEL
LIN {X 0,Y 361.381,Z 401.97,A -85,B 0,C 180,E1 -13145.58,E2 -13145.58} C_VEL
LIN {X 0,Y 361.594,Z 397.043,A -85,B 0,C 180,E1 -13147.329,E2 -13147.329} C_VEL
LIN {X 0,Y 361.957,Z 391.317,A -85,B 0,C 180,E1 -13148.936,E2 -13148.936} C_VEL
LIN {X 0,Y 362.531,Z 383.904,A -85,B 0,C 180,E1 -13150.613,E2 -13150.613} C_VEL
LIN {X 0,Y 363.181,Z 374.679,A -85,B 0,C 180,E1 -13152.29,E2 -13152.29} C_VEL
LIN {X 0,Y 363.924,Z 365.283,A -85,B 0,C 180,E1 -13153.684,E2 -13153.684} C_VEL
LIN {X 0,Y 364.699,Z 353.837,A -85,B 0,C 180,E1 -13155.057,E2 -13155.057} C_VEL
LIN {X 0,Y 365.371,Z 342.079,A -85,B 0,C 180,E1 -13156.195,E2 -13156.195} C_VEL
LIN {X 0,Y 366.03,Z 329.872,A -85,B 0,C 180,E1 -13157.119,E2 -13157.119} C_VEL
LIN {X 0,Y 366.199,Z 326.1,A -85,B 0,C 180,E1 -13157.364,E2 -13157.364} C_VEL
LIN {X 0,Y 362.895,Z 311.536,A -85,B 0,C 180,E1 -13158.268,E2 -13158.268} C_VEL
LIN {X 0,Y 361.193,Z 304.497,A -85,B 0,C 180,E1 -13158.616,E2 -13158.616} C_VEL
LIN {X 0,Y 361.506,Z 304.449,A -85,B 0,C 180,E1 -13161.677,E2 -13161.677} C_VEL
LIN {X 0,Y 361.743,Z 304.427,A -85,B 0,C 180,E1 -13164.079,E2 -13164.079} C_VEL
LIN {X 0,Y 361.883,Z 304.4,A -85,B 0,C 180,E1 -13166.702,E2 -13166.702} C_VEL
LIN {X 0,Y 361.875,Z 304.406,A -85,B 0,C 180,E1 -13170.328,E2 -13170.328} C_VEL
LIN {X 0,Y 361.857,Z 304.41,A -85,B 0,C 180,E1 -13174.28,E2 -13174.28} C_VEL
LIN {X 0,Y 361.866,Z 304.411,A -85,B 0,C 180,E1 -13177.223,E2 -13177.223} C_VEL
LIN {X 0,Y 361.838,Z 304.415,A -85,B 0,C 180,E1 -13180.755,E2 -13180.755} C_VEL
LIN {X 0,Y 361.82,Z 304.414,A -85,B 0,C 180,E1 -13184.368,E2 -13184.368} C_VEL
LIN {X 0,Y 361.838,Z 304.414,A -85,B 0,C 180,E1 -13187.568,E2 -13187.568} C_VEL
LIN {X 0,Y 361.871,Z 304.409,A -85,B 0,C 180,E1 -13190.973,E2 -13190.973} C_VEL
LIN {X 0,Y 361.803,Z 304.421,A -85,B 0,C 180,E1 -13194.356,E2 -13194.356} C_VEL
LIN {X 0,Y 361.774,Z 304.539,A -85,B 0,C 180,E1 -13195.842,E2 -13195.842} C_VEL
LIN {X 0,Y 361.569,Z 309.094,A -85,B 0,C 180,E1 -13198.788,E2 -13198.788} C_VEL
LIN {X 0,Y 361.447,Z 314.38,A -85,B 0,C 180,E1 -13202.182,E2 -13202.182} C_VEL
LIN {X 0,Y 361.35,Z 320.654,A -85,B 0,C 180,E1 -13206.081,E2 -13206.081} C_VEL
LIN {X 0,Y 361.359,Z 326.522,A -85,B 0,C 180,E1 -13209.508,E2 -13209.508} C_VEL
LIN {X 0,Y 361.338,Z 327.519,A -85,B 0,C 180,E1 -13210.042,E2 -13210.042} C_VEL
LIN {X 0,Y 365.068,Z 341.024,A -85,B 0,C 180,E1 -13210.73,E2 -13210.73} C_VEL
LIN {X 0,Y 367.676,Z 352.693,A -85,B 0,C 180,E1 -13211.496,E2 -13211.496} C_VEL
LIN {X 0,Y 368.05,Z 356.611,A -85,B 0,C 180,E1 -13211.777,E2 -13211.777} C_VEL
LIN {X 0,Y 367.234,Z 367.725,A -85,B 0,C 180,E1 -13212.601,E2 -13212.601} C_VEL
LIN {X 0,Y 366.36,Z 377.987,A -85,B 0,C 180,E1 -13213.571,E2 -13213.571} C_VEL
LIN {X 0,Y 365.477,Z 388.382,A -85,B 0,C 180,E1 -13214.811,E2 -13214.811} C_VEL
LIN {X 0,Y 364.337,Z 398.691,A -85,B 0,C 180,E1 -13216.332,E2 -13216.332} C_VEL
LIN {X 0,Y 363.297,Z 407.612,A -85,B 0,C 180,E1 -13217.997,E2 -13217.997} C_VEL
LIN {X 0,Y 362.44,Z 414.776,A -85,B 0,C 180,E1 -13219.667,E2 -13219.667} C_VEL
LIN {X 0,Y 361.702,Z 421.336,A -85,B 0,C 180,E1 -13221.621,E2 -13221.621} C_VEL
LIN {X 0,Y 361.303,Z 425.641,A -85,B 0,C 180,E1 -13223.298,E2 -13223.298} C_VEL
LIN {X 0,Y 360.963,Z 427.915,A -85,B 0,C 180,E1 -13224.413,E2 -13224.413} C_VEL
LIN {X 0,Y 360.849,Z 429.76,A -85,B 0,C 180,E1 -13225.532,E2 -13225.532} C_VEL
LIN {X 0,Y 360.833,Z 431.163,A -85,B 0,C 180,E1 -13226.65,E2 -13226.65} C_VEL
LIN {X 0,Y 360.564,Z 432.77,A -85,B 0,C 180,E1 -13228.883,E2 -13228.883} C_VEL
LIN {X 0,Y 360.537,Z 433.004,A -85,B 0,C 180,E1 -13230,E2 -13230} C_VEL
LIN {X 0,Y 360.684,Z 432.225,A -85,B 0,C 180,E1 -13232.233,E2 -13232.233} C_VEL
LIN {X 0,Y 360.81,Z 431.262,A -85,B 0,C 180,E1 -13233.35,E2 -13233.35} C_VEL
LIN {X 0,Y 360.822,Z 429.913,A -85,B 0,C 180,E1 -13234.469,E2 -13234.469} C_VEL
LIN {X 0,Y 361.113,Z 427.058,A -85,B 0,C 180,E1 -13236.145,E2 -13236.145} C_VEL
LIN {X 0,Y 361.515,Z 423.18,A -85,B 0,C 180,E1 -13237.821,E2 -13237.821} C_VEL
LIN {X 0,Y 362.041,Z 418.157,A -85,B 0,C 180,E1 -13239.497,E2 -13239.497} C_VEL
LIN {X 0,Y 362.861,Z 411.807,A -85,B 0,C 180,E1 -13241.168,E2 -13241.168} C_VEL
LIN {X 0,Y 363.761,Z 403.919,A -85,B 0,C 180,E1 -13242.837,E2 -13242.837} C_VEL
LIN {X 0,Y 364.709,Z 395.851,A -85,B 0,C 180,E1 -13244.223,E2 -13244.223} C_VEL
LIN {X 0,Y 365.728,Z 385.945,A -85,B 0,C 180,E1 -13245.607,E2 -13245.607} C_VEL
LIN {X 0,Y 366.53,Z 376.161,A -85,B 0,C 180,E1 -13246.715,E2 -13246.715} C_VEL
LIN {X 0,Y 367.464,Z 365.533,A -85,B 0,C 180,E1 -13247.675,E2 -13247.675} C_VEL
LIN {X 0,Y 368.085,Z 354.69,A -85,B 0,C 180,E1 -13248.453,E2 -13248.453} C_VEL
LIN {X 0,Y 365.397,Z 342.379,A -85,B 0,C 180,E1 -13249.295,E2 -13249.295} C_VEL
LIN {X 0,Y 361.933,Z 329.714,A -85,B 0,C 180,E1 -13249.965,E2 -13249.965} C_VEL
LIN {X 0,Y 361.353,Z 327.442,A -85,B 0,C 180,E1 -13250.089,E2 -13250.089} C_VEL
LIN {X 0,Y 361.359,Z 322.558,A -85,B 0,C 180,E1 -13252.891,E2 -13252.891} C_VEL
LIN {X 0,Y 361.4,Z 316.542,A -85,B 0,C 180,E1 -13256.569,E2 -13256.569} C_VEL
LIN {X 0,Y 361.442,Z 313.674,A -85,B 0,C 180,E1 -13258.395,E2 -13258.395} C_VEL
LIN {X 0,Y 360.83,Z 312.351,A -85,B 0,C 180,E1 -13259.302,E2 -13259.302} C_VEL
LIN {X 0,Y 358.098,Z 310.502,A -85,B 0,C 180,E1 -13260.792,E2 -13260.792} C_VEL
LIN {X 0,Y 355.785,Z 309.044,A -85,B 0,C 180,E1 -13261.997,E2 -13261.997} C_VEL
LIN {X 0,Y 354.814,Z 307.79,A -85,B 0,C 180,E1 -13262.923,E2 -13262.923} C_VEL
LIN {X 0,Y 354.747,Z 307.311,A -85,B 0,C 180,E1 -13263.234,E2 -13263.234} C_VEL
LIN {X 0,Y 354.77,Z 305.296,A -85,B 0,C 180,E1 -13264.545,E2 -13264.545} C_VEL
LIN {X 0,Y 354.803,Z 305.291,A -85,B 0,C 180,E1 -13267.883,E2 -13267.883} C_VEL
LIN {X 0,Y 354.79,Z 305.294,A -85,B 0,C 180,E1 -13271.172,E2 -13271.172} C_VEL
LIN {X 0,Y 354.766,Z 305.297,A -85,B 0,C 180,E1 -13274.506,E2 -13274.506} C_VEL
LIN {X 0,Y 354.796,Z 305.292,A -85,B 0,C 180,E1 -13277.663,E2 -13277.663} C_VEL
LIN {X 0,Y 354.817,Z 305.288,A -85,B 0,C 180,E1 -13280.666,E2 -13280.666} C_VEL
LIN {X 0,Y 354.729,Z 305.297,A -85,B 0,C 180,E1 -13284.322,E2 -13284.322} C_VEL
LIN {X 0,Y 354.546,Z 305.44,A -85,B 0,C 180,E1 -13287.052,E2 -13287.052} C_VEL
LIN {X 0,Y 354.192,Z 312.55,A -85,B 0,C 180,E1 -13291.561,E2 -13291.561} C_VEL
LIN {X 0,Y 354.132,Z 316.571,A -85,B 0,C 180,E1 -13294.112,E2 -13294.112} C_VEL
LIN {X 0,Y 354.085,Z 320.468,A -85,B 0,C 180,E1 -13296.611,E2 -13296.611} C_VEL
LIN {X 0,Y 354,Z 326.432,A -85,B 0,C 180,E1 -13300.275,E2 -13300.275} C_VEL
LIN {X 0,Y 354.029,Z 328.194,A -85,B 0,C 180,E1 -13301.256,E2 -13301.256} C_VEL
LIN {X 0,Y 356.538,Z 340.62,A -85,B 0,C 180,E1 -13301.872,E2 -13301.872} C_VEL
LIN {X 0,Y 358.697,Z 352.007,A -85,B 0,C 180,E1 -13302.61,E2 -13302.61} C_VEL
LIN {X 0,Y 358.086,Z 365.45,A -85,B 0,C 180,E1 -13303.612,E2 -13303.612} C_VEL
LIN {X 0,Y 357.344,Z 376.708,A -85,B 0,C 180,E1 -13304.687,E2 -13304.687} C_VEL
LIN {X 0,Y 356.587,Z 388.061,A -85,B 0,C 180,E1 -13306.029,E2 -13306.029} C_VEL
LIN {X 0,Y 355.743,Z 397.785,A -85,B 0,C 180,E1 -13307.449,E2 -13307.449} C_VEL
LIN {X 0,Y 355.071,Z 407.322,A -85,B 0,C 180,E1 -13309.162,E2 -13309.162} C_VEL
LIN {X 0,Y 354.485,Z 414.941,A -85,B 0,C 180,E1 -13310.874,E2 -13310.874} C_VEL
LIN {X 0,Y 354.051,Z 421.284,A -85,B 0,C 180,E1 -13312.644,E2 -13312.644} C_VEL
LIN {X 0,Y 353.803,Z 425.949,A -85,B 0,C 180,E1 -13314.3,E2 -13314.3} C_VEL
LIN {X 0,Y 353.642,Z 429.619,A -85,B 0,C 180,E1 -13316.011,E2 -13316.011} C_VEL
LIN {X 0,Y 353.586,Z 432.223,A -85,B 0,C 180,E1 -13317.722,E2 -13317.722} C_VEL
LIN {X 0,Y 353.517,Z 433.389,A -85,B 0,C 180,E1 -13318.861,E2 -13318.861} C_VEL
LIN {X 0,Y 353.5,Z 434.144,A -85,B 0,C 180,E1 -13320,E2 -13320} C_VEL
LIN {X 0,Y 353.551,Z 434.458,A -85,B 0,C 180,E1 -13321.139,E2 -13321.139} C_VEL
LIN {X 0,Y 353.683,Z 434.316,A -85,B 0,C 180,E1 -13322.278,E2 -13322.278} C_VEL
LIN {X 0,Y 353.871,Z 433.771,A -85,B 0,C 180,E1 -13323.416,E2 -13323.416} C_VEL
LIN {X 0,Y 354.098,Z 432.782,A -85,B 0,C 180,E1 -13324.553,E2 -13324.553} C_VEL
LIN {X 0,Y 354.232,Z 431.346,A -85,B 0,C 180,E1 -13325.693,E2 -13325.693} C_VEL
LIN {X 0,Y 354.56,Z 428.556,A -85,B 0,C 180,E1 -13327.299,E2 -13327.299} C_VEL
LIN {X 0,Y 355.333,Z 424.239,A -85,B 0,C 180,E1 -13329.104,E2 -13329.104} C_VEL
LIN {X 0,Y 356.001,Z 418.961,A -85,B 0,C 180,E1 -13330.81,E2 -13330.81} C_VEL
LIN {X 0,Y 356.972,Z 412.243,A -85,B 0,C 180,E1 -13332.507,E2 -13332.507} C_VEL
LIN {X 0,Y 358.201,Z 403.891,A -85,B 0,C 180,E1 -13334.197,E2 -13334.197} C_VEL
LIN {X 0,Y 359.387,Z 395.412,A -85,B 0,C 180,E1 -13335.598,E2 -13335.598} C_VEL
LIN {X 0,Y 360.812,Z 383.747,A -85,B 0,C 180,E1 -13337.156,E2 -13337.156} C_VEL
LIN {X 0,Y 362.319,Z 370.649,A -85,B 0,C 180,E1 -13338.52,E2 -13338.52} C_VEL
LIN {X 0,Y 363.439,Z 358.782,A -85,B 0,C 180,E1 -13339.493,E2 -13339.493} C_VEL
LIN {X 0,Y 360.989,Z 348.516,A -85,B 0,C 180,E1 -13340.468,E2 -13340.468} C_VEL
LIN {X 0,Y 357.263,Z 337.889,A -85,B 0,C 180,E1 -13341.478,E2 -13341.478} C_VEL
LIN {X 0,Y 355.494,Z 333.365,A -85,B 0,C 180,E1 -13341.919,E2 -13341.919} C_VEL
LIN {X 0,Y 355.747,Z 329.105,A -85,B 0,C 180,E1 -13344.665,E2 -13344.665} C_VEL
LIN {X 0,Y 356.184,Z 322.496,A -85,B 0,C 180,E1 -13348.909,E2 -13348.909} C_VEL
LIN {X 0,Y 356.766,Z 316.439,A -85,B 0,C 180,E1 -13352.801,E2 -13352.801} C_VEL
LIN {X 0,Y 356.607,Z 313.465,A -85,B 0,C 180,E1 -13354.857,E2 -13354.857} C_VEL
LIN {X 0,Y 355.874,Z 309.531,A -85,B 0,C 180,E1 -13357.82,E2 -13357.82} C_VEL
LIN {X 0,Y 354.78,Z 305.3,A -85,B 0,C 180,E1 -13361.494,E2 -13361.494} C_VEL
LIN {X 0,Y 354.817,Z 305.306,A -85,B 0,C 180,E1 -13362.616,E2 -13362.616} C_VEL
LIN {X 0,Y 356.168,Z 312.434,A -85,B 0,C 180,E1 -13366.32,E2 -13366.32} C_VEL
LIN {X 0,Y 357.626,Z 319.958,A -85,B 0,C 180,E1 -13370.034,E2 -13370.034} C_VEL
LIN {X 0,Y 358.54,Z 325.368,A -85,B 0,C 180,E1 -13372.58,E2 -13372.58} C_VEL
LIN {X 0,Y 358.411,Z 328.494,A -85,B 0,C 180,E1 -13373.966,E2 -13373.966} C_VEL
LIN {X 0,Y 357.3,Z 337.734,A -85,B 0,C 180,E1 -13377.921,E2 -13377.921} C_VEL
LIN {X 0,Y 356.446,Z 345.388,A -85,B 0,C 180,E1 -13381.114,E2 -13381.114} C_VEL
LIN {X 0,Y 355.631,Z 354.54,A -85,B 0,C 180,E1 -13384.857,E2 -13384.857} C_VEL
LIN {X 0,Y 354.839,Z 364.505,A -85,B 0,C 180,E1 -13388.818,E2 -13388.818} C_VEL
LIN {X 0,Y 357.478,Z 378.085,A -85,B 0,C 180,E1 -13389.668,E2 -13389.668} C_VEL
LIN {X 0,Y 358.671,Z 390.726,A -85,B 0,C 180,E1 -13390.542,E2 -13390.542} C_VEL
LIN {X 0,Y 359.707,Z 404.113,A -85,B 0,C 180,E1 -13391.679,E2 -13391.679} C_VEL
LIN {X 0,Y 359.422,Z 409.921,A -85,B 0,C 180,E1 -13392.21,E2 -13392.21} C_VEL
LIN {X 0,Y 358.04,Z 421.917,A -85,B 0,C 180,E1 -13393.464,E2 -13393.464} C_VEL
LIN {X 0,Y 356.884,Z 432.083,A -85,B 0,C 180,E1 -13394.784,E2 -13394.784} C_VEL
LIN {X 0,Y 355.871,Z 441.532,A -85,B 0,C 180,E1 -13396.291,E2 -13396.291} C_VEL
LIN {X 0,Y 354.915,Z 450.298,A -85,B 0,C 180,E1 -13397.999,E2 -13397.999} C_VEL
LIN {X 0,Y 354.27,Z 457.382,A -85,B 0,C 180,E1 -13399.715,E2 -13399.715} C_VEL
LIN {X 0,Y 353.806,Z 463.081,A -85,B 0,C 180,E1 -13401.432,E2 -13401.432} C_VEL
LIN {X 0,Y 353.59,Z 467.58,A -85,B 0,C 180,E1 -13403.151,E2 -13403.151} C_VEL
LIN {X 0,Y 353.484,Z 469.975,A -85,B 0,C 180,E1 -13404.295,E2 -13404.295} C_VEL
LIN {X 0,Y 353.408,Z 471.891,A -85,B 0,C 180,E1 -13405.438,E2 -13405.438} C_VEL
LIN {X 0,Y 353.381,Z 473.342,A -85,B 0,C 180,E1 -13406.579,E2 -13406.579} C_VEL
LIN {X 0,Y 353.401,Z 474.383,A -85,B 0,C 180,E1 -13407.721,E2 -13407.721} C_VEL
LIN {X 0,Y 353.537,Z 474.998,A -85,B 0,C 180,E1 -13408.861,E2 -13408.861} C_VEL
LIN {X 0,Y 353.534,Z 475.141,A -85,B 0,C 180,E1 -13410,E2 -13410} C_VEL
LIN {X 0,Y 353.534,Z 474.873,A -85,B 0,C 180,E1 -13411.139,E2 -13411.139} C_VEL
LIN {X 0,Y 353.431,Z 474.178,A -85,B 0,C 180,E1 -13412.279,E2 -13412.279} C_VEL
LIN {X 0,Y 353.435,Z 471.481,A -85,B 0,C 180,E1 -13414.562,E2 -13414.562} C_VEL
LIN {X 0,Y 353.536,Z 468.415,A -85,B 0,C 180,E1 -13416.301,E2 -13416.301} C_VEL
LIN {X 0,Y 353.688,Z 464.372,A -85,B 0,C 180,E1 -13417.995,E2 -13417.995} C_VEL
LIN {X 0,Y 354.163,Z 458.07,A -85,B 0,C 180,E1 -13419.999,E2 -13419.999} C_VEL
LIN {X 0,Y 354.773,Z 451.198,A -85,B 0,C 180,E1 -13421.715,E2 -13421.715} C_VEL
LIN {X 0,Y 355.709,Z 442.607,A -85,B 0,C 180,E1 -13423.424,E2 -13423.424} C_VEL
LIN {X 0,Y 356.819,Z 432.307,A -85,B 0,C 180,E1 -13425.177,E2 -13425.177} C_VEL
LIN {X 0,Y 358.152,Z 421.351,A -85,B 0,C 180,E1 -13426.678,E2 -13426.678} C_VEL
LIN {X 0,Y 359.618,Z 410.131,A -85,B 0,C 180,E1 -13427.927,E2 -13427.927} C_VEL
LIN {X 0,Y 359.944,Z 404.364,A -85,B 0,C 180,E1 -13428.499,E2 -13428.499} C_VEL
LIN {X 0,Y 359.393,Z 392.534,A -85,B 0,C 180,E1 -13429.582,E2 -13429.582} C_VEL
LIN {X 0,Y 358.517,Z 380.187,A -85,B 0,C 180,E1 -13430.533,E2 -13430.533} C_VEL
LIN {X 0,Y 356.335,Z 367.539,A -85,B 0,C 180,E1 -13431.431,E2 -13431.431} C_VEL
LIN {X 0,Y 354.79,Z 360.663,A -85,B 0,C 180,E1 -13431.926,E2 -13431.926} C_VEL
LIN {X 0,Y 355.467,Z 352.78,A -85,B 0,C 180,E1 -13435.156,E2 -13435.156} C_VEL
LIN {X 0,Y 356.287,Z 344.115,A -85,B 0,C 180,E1 -13438.9,E2 -13438.9} C_VEL
LIN {X 0,Y 357.27,Z 336.91,A -85,B 0,C 180,E1 -13442.235,E2 -13442.235} C_VEL
LIN {X 0,Y 358.562,Z 329.482,A -85,B 0,C 180,E1 -13446.016,E2 -13446.016} C_VEL
LIN {X 0,Y 358.835,Z 327.084,A -85,B 0,C 180,E1 -13447.384,E2 -13447.384} C_VEL
LIN {X 0,Y 358.275,Z 323.058,A -85,B 0,C 180,E1 -13450.09,E2 -13450.09} C_VEL
LIN {X 0,Y 357.501,Z 318.975,A -85,B 0,C 180,E1 -13453.477,E2 -13453.477} C_VEL
LIN {X 0,Y 356.931,Z 315.979,A -85,B 0,C 180,E1 -13456.764,E2 -13456.764} C_VEL
LIN {X 0,Y 356.532,Z 313.853,A -85,B 0,C 180,E1 -13460.244,E2 -13460.244} C_VEL
LIN {X 0,Y 356.358,Z 313.063,A -85,B 0,C 180,E1 -13462.311,E2 -13462.311} C_VEL
LIN {X 0,Y 356.186,Z 312.427,A -85,B 0,C 180,E1 -13465.967,E2 -13465.967} C_VEL
LIN {X 0,Y 356.139,Z 312.565,A -85,B 0,C 180,E1 -13469.131,E2 -13469.131} C_VEL
LIN {X 0,Y 356.232,Z 313.413,A -85,B 0,C 180,E1 -13473.015,E2 -13473.015} C_VEL
LIN {X 0,Y 356.197,Z 314.324,A -85,B 0,C 180,E1 -13475.522,E2 -13475.522} C_VEL
LIN {X 0,Y 356.035,Z 315.575,A -85,B 0,C 180,E1 -13478.223,E2 -13478.223} C_VEL
LIN {X 0,Y 357.331,Z 318.567,A -85,B 0,C 180,E1 -13478.538,E2 -13478.538} C_VEL
LIN {X 0,Y 361.726,Z 328.497,A -85,B 0,C 180,E1 -13479.627,E2 -13479.627} C_VEL
LIN {X 0,Y 364.318,Z 336.139,A -85,B 0,C 180,E1 -13480.452,E2 -13480.452} C_VEL
LIN {X 0,Y 364.142,Z 340.989,A -85,B 0,C 180,E1 -13480.846,E2 -13480.846} C_VEL
LIN {X 0,Y 362.885,Z 353.125,A -85,B 0,C 180,E1 -13481.948,E2 -13481.948} C_VEL
LIN {X 0,Y 361.599,Z 364.08,A -85,B 0,C 180,E1 -13483.195,E2 -13483.195} C_VEL
LIN {X 0,Y 360.179,Z 374.904,A -85,B 0,C 180,E1 -13484.727,E2 -13484.727} C_VEL
LIN {X 0,Y 359.019,Z 382.905,A -85,B 0,C 180,E1 -13486.125,E2 -13486.125} C_VEL
LIN {X 0,Y 357.846,Z 390.708,A -85,B 0,C 180,E1 -13487.812,E2 -13487.812} C_VEL
LIN {X 0,Y 357.008,Z 396.06,A -85,B 0,C 180,E1 -13489.221,E2 -13489.221} C_VEL
LIN {X 0,Y 356.084,Z 401.235,A -85,B 0,C 180,E1 -13490.915,E2 -13490.915} C_VEL
LIN {X 0,Y 355.387,Z 405.205,A -85,B 0,C 180,E1 -13492.615,E2 -13492.615} C_VEL
LIN {X 0,Y 354.937,Z 408.089,A -85,B 0,C 180,E1 -13494.318,E2 -13494.318} C_VEL
LIN {X 0,Y 354.603,Z 409.48,A -85,B 0,C 180,E1 -13495.453,E2 -13495.453} C_VEL
LIN {X 0,Y 354.246,Z 410.427,A -85,B 0,C 180,E1 -13496.588,E2 -13496.588} C_VEL
LIN {X 0,Y 353.988,Z 410.925,A -85,B 0,C 180,E1 -13497.724,E2 -13497.724} C_VEL
LIN {X 0,Y 353.85,Z 411.009,A -85,B 0,C 180,E1 -13498.862,E2 -13498.862} C_VEL
LIN {X 0,Y 353.798,Z 410.675,A -85,B 0,C 180,E1 -13500,E2 -13500} C_VEL
LIN {X 0,Y 353.829,Z 409.875,A -85,B 0,C 180,E1 -13501.138,E2 -13501.138} C_VEL
LIN {X 0,Y 353.914,Z 408.665,A -85,B 0,C 180,E1 -13502.276,E2 -13502.276} C_VEL
LIN {X 0,Y 354.138,Z 406.028,A -85,B 0,C 180,E1 -13503.983,E2 -13503.983} C_VEL
LIN {X 0,Y 354.308,Z 402.359,A -85,B 0,C 180,E1 -13505.692,E2 -13505.692} C_VEL
LIN {X 0,Y 354.595,Z 396.622,A -85,B 0,C 180,E1 -13507.695,E2 -13507.695} C_VEL
LIN {X 0,Y 355.024,Z 390.311,A -85,B 0,C 180,E1 -13509.4,E2 -13509.4} C_VEL
LIN {X 0,Y 355.629,Z 382.467,A -85,B 0,C 180,E1 -13511.109,E2 -13511.109} C_VEL
LIN {X 0,Y 356.202,Z 374.517,A -85,B 0,C 180,E1 -13512.535,E2 -13512.535} C_VEL
LIN {X 0,Y 357.066,Z 363.827,A -85,B 0,C 180,E1 -13514.098,E2 -13514.098} C_VEL
LIN {X 0,Y 357.855,Z 352.123,A -85,B 0,C 180,E1 -13515.48,E2 -13515.48} C_VEL
LIN {X 0,Y 358.569,Z 339.475,A -85,B 0,C 180,E1 -13516.658,E2 -13516.658} C_VEL
LIN {X 0,Y 359.255,Z 327.865,A -85,B 0,C 180,E1 -13517.508,E2 -13517.508} C_VEL
LIN {X 0,Y 356.998,Z 317.205,A -85,B 0,C 180,E1 -13518.22,E2 -13518.22} C_VEL
LIN {X 0,Y 354.193,Z 305.368,A -85,B 0,C 180,E1 -13518.863,E2 -13518.863} C_VEL
LIN {X 0,Y 354.492,Z 305.324,A -85,B 0,C 180,E1 -13522.129,E2 -13522.129} C_VEL
LIN {X 0,Y 354.718,Z 305.302,A -85,B 0,C 180,E1 -13524.587,E2 -13524.587} C_VEL
LIN {X 0,Y 354.823,Z 305.281,A -85,B 0,C 180,E1 -13527.101,E2 -13527.101} C_VEL
LIN {X 0,Y 354.82,Z 305.285,A -85,B 0,C 180,E1 -13529.682,E2 -13529.682} C_VEL
LIN {X 0,Y 354.808,Z 305.289,A -85,B 0,C 180,E1 -13533.702,E2 -13533.702} C_VEL
LIN {X 0,Y 354.801,Z 305.292,A -85,B 0,C 180,E1 -13536.459,E2 -13536.459} C_VEL
LIN {X 0,Y 354.826,Z 305.285,A -85,B 0,C 180,E1 -13539.424,E2 -13539.424} C_VEL
LIN {X 0,Y 354.791,Z 305.292,A -85,B 0,C 180,E1 -13542.867,E2 -13542.867} C_VEL
LIN {X 0,Y 354.77,Z 305.294,A -85,B 0,C 180,E1 -13546.104,E2 -13546.104} C_VEL
LIN {X 0,Y 354.79,Z 305.291,A -85,B 0,C 180,E1 -13549.179,E2 -13549.179} C_VEL
LIN {X 0,Y 354.803,Z 305.289,A -85,B 0,C 180,E1 -13552.404,E2 -13552.404} C_VEL
LIN {X 0,Y 354.771,Z 305.371,A -85,B 0,C 180,E1 -13555.627,E2 -13555.627} C_VEL
LIN {X 0,Y 354.564,Z 309.725,A -85,B 0,C 180,E1 -13558.466,E2 -13558.466} C_VEL
LIN {X 0,Y 354.431,Z 315.557,A -85,B 0,C 180,E1 -13562.226,E2 -13562.226} C_VEL
LIN {X 0,Y 354.325,Z 321.351,A -85,B 0,C 180,E1 -13565.84,E2 -13565.84} C_VEL
LIN {X 0,Y 354.34,Z 327.405,A -85,B 0,C 180,E1 -13569.387,E2 -13569.387} C_VEL
LIN {X 0,Y 354.343,Z 327.833,A -85,B 0,C 180,E1 -13569.627,E2 -13569.627} C_VEL
LIN {X 0,Y 358.189,Z 341.699,A -85,B 0,C 180,E1 -13570.358,E2 -13570.358} C_VEL
LIN {X 0,Y 360.938,Z 354.126,A -85,B 0,C 180,E1 -13571.205,E2 -13571.205} C_VEL
LIN {X 0,Y 361.312,Z 357.315,A -85,B 0,C 180,E1 -13571.446,E2 -13571.446} C_VEL
LIN {X 0,Y 360.363,Z 369.71,A -85,B 0,C 180,E1 -13572.405,E2 -13572.405} C_VEL
LIN {X 0,Y 359.34,Z 380.516,A -85,B 0,C 180,E1 -13573.489,E2 -13573.489} C_VEL
LIN {X 0,Y 358.427,Z 390.864,A -85,B 0,C 180,E1 -13574.796,E2 -13574.796} C_VEL
LIN {X 0,Y 357.454,Z 399.103,A -85,B 0,C 180,E1 -13576.063,E2 -13576.063} C_VEL
LIN {X 0,Y 356.378,Z 408.025,A -85,B 0,C 180,E1 -13577.761,E2 -13577.761} C_VEL
LIN {X 0,Y 355.476,Z 415.189,A -85,B 0,C 180,E1 -13579.462,E2 -13579.462} C_VEL
LIN {X 0,Y 354.706,Z 421.75,A -85,B 0,C 180,E1 -13581.454,E2 -13581.454} C_VEL
LIN {X 0,Y 354.257,Z 426.057,A -85,B 0,C 180,E1 -13583.164,E2 -13583.164} C_VEL
LIN {X 0,Y 353.926,Z 428.329,A -85,B 0,C 180,E1 -13584.302,E2 -13584.302} C_VEL
LIN {X 0,Y 353.773,Z 430.176,A -85,B 0,C 180,E1 -13585.442,E2 -13585.442} C_VEL
LIN {X 0,Y 353.761,Z 431.578,A -85,B 0,C 180,E1 -13586.583,E2 -13586.583} C_VEL
LIN {X 0,Y 353.501,Z 433.184,A -85,B 0,C 180,E1 -13588.861,E2 -13588.861} C_VEL
LIN {X 0,Y 353.471,Z 433.418,A -85,B 0,C 180,E1 -13590,E2 -13590} C_VEL
LIN {X 0,Y 353.627,Z 432.638,A -85,B 0,C 180,E1 -13592.278,E2 -13592.278} C_VEL
LIN {X 0,Y 353.739,Z 431.675,A -85,B 0,C 180,E1 -13593.417,E2 -13593.417} C_VEL
LIN {X 0,Y 353.747,Z 430.327,A -85,B 0,C 180,E1 -13594.558,E2 -13594.558} C_VEL
LIN {X 0,Y 354.087,Z 427.47,A -85,B 0,C 180,E1 -13596.267,E2 -13596.267} C_VEL
LIN {X 0,Y 354.484,Z 423.593,A -85,B 0,C 180,E1 -13597.977,E2 -13597.977} C_VEL
LIN {X 0,Y 355.038,Z 418.569,A -85,B 0,C 180,E1 -13599.687,E2 -13599.687} C_VEL
LIN {X 0,Y 355.911,Z 412.217,A -85,B 0,C 180,E1 -13601.389,E2 -13601.389} C_VEL
LIN {X 0,Y 356.863,Z 404.326,A -85,B 0,C 180,E1 -13603.09,E2 -13603.09} C_VEL
LIN {X 0,Y 357.852,Z 396.255,A -85,B 0,C 180,E1 -13604.501,E2 -13604.501} C_VEL
LIN {X 0,Y 358.91,Z 386.345,A -85,B 0,C 180,E1 -13605.911,E2 -13605.911} C_VEL
LIN {X 0,Y 359.746,Z 376.556,A -85,B 0,C 180,E1 -13607.04,E2 -13607.04} C_VEL
LIN {X 0,Y 360.739,Z 365.92,A -85,B 0,C 180,E1 -13608.016,E2 -13608.016} C_VEL
LIN {X 0,Y 361.359,Z 356.635,A -85,B 0,C 180,E1 -13608.702,E2 -13608.702} C_VEL
LIN {X 0,Y 358.978,Z 345.045,A -85,B 0,C 180,E1 -13609.537,E2 -13609.537} C_VEL
LIN {X 0,Y 355.639,Z 332.418,A -85,B 0,C 180,E1 -13610.265,E2 -13610.265} C_VEL
LIN {X 0,Y 354.358,Z 327.824,A -85,B 0,C 180,E1 -13610.495,E2 -13610.495} C_VEL
LIN {X 0,Y 354.331,Z 322.847,A -85,B 0,C 180,E1 -13613.372,E2 -13613.372} C_VEL
LIN {X 0,Y 354.378,Z 316.735,A -85,B 0,C 180,E1 -13617.138,E2 -13617.138} C_VEL
LIN {X 0,Y 354.518,Z 311.702,A -85,B 0,C 180,E1 -13620.366,E2 -13620.366} C_VEL
LIN {X 0,Y 354.747,Z 307.311,A -85,B 0,C 180,E1 -13623.234,E2 -13623.234} C_VEL
LIN {X 0,Y 354.113,Z 306.248,A -85,B 0,C 180,E1 -13624.163,E2 -13624.163} C_VEL
LIN {X 0,Y 352.564,Z 305.813,A -85,B 0,C 180,E1 -13625.089,E2 -13625.089} C_VEL
LIN {X 0,Y 348.896,Z 306.028,A -85,B 0,C 180,E1 -13626.959,E2 -13626.959} C_VEL
LIN {X 0,Y 347.85,Z 306.158,A -85,B 0,C 180,E1 -13627.93,E2 -13627.93} C_VEL
LIN {X 0,Y 347.758,Z 306.167,A -85,B 0,C 180,E1 -13628.259,E2 -13628.259} C_VEL
LIN {X 0,Y 347.753,Z 306.169,A -85,B 0,C 180,E1 -13631.83,E2 -13631.83} C_VEL
LIN {X 0,Y 347.708,Z 306.177,A -85,B 0,C 180,E1 -13635.027,E2 -13635.027} C_VEL
LIN {X 0,Y 347.753,Z 306.167,A -85,B 0,C 180,E1 -13638.397,E2 -13638.397} C_VEL
LIN {X 0,Y 347.766,Z 306.163,A -85,B 0,C 180,E1 -13642.013,E2 -13642.013} C_VEL
LIN {X 0,Y 347.606,Z 306.181,A -85,B 0,C 180,E1 -13645.52,E2 -13645.52} C_VEL
LIN {X 0,Y 347.49,Z 306.405,A -85,B 0,C 180,E1 -13647.092,E2 -13647.092} C_VEL
LIN {X 0,Y 347.149,Z 313.463,A -85,B 0,C 180,E1 -13651.591,E2 -13651.591} C_VEL
LIN {X 0,Y 347.05,Z 318.508,A -85,B 0,C 180,E1 -13654.832,E2 -13654.832} C_VEL
LIN {X 0,Y 346.973,Z 323.517,A -85,B 0,C 180,E1 -13657.993,E2 -13657.993} C_VEL
LIN {X 0,Y 346.948,Z 328.325,A -85,B 0,C 180,E1 -13660.993,E2 -13660.993} C_VEL
LIN {X 0,Y 349.455,Z 340.937,A -85,B 0,C 180,E1 -13661.636,E2 -13661.636} C_VEL
LIN {X 0,Y 351.777,Z 353.508,A -85,B 0,C 180,E1 -13662.479,E2 -13662.479} C_VEL
LIN {X 0,Y 351.109,Z 365.872,A -85,B 0,C 180,E1 -13663.427,E2 -13663.427} C_VEL
LIN {X 0,Y 350.366,Z 376.957,A -85,B 0,C 180,E1 -13664.505,E2 -13664.505} C_VEL
LIN {X 0,Y 349.563,Z 388.485,A -85,B 0,C 180,E1 -13665.89,E2 -13665.89} C_VEL
LIN {X 0,Y 348.646,Z 399.101,A -85,B 0,C 180,E1 -13667.485,E2 -13667.485} C_VEL
LIN {X 0,Y 348.056,Z 407.047,A -85,B 0,C 180,E1 -13668.941,E2 -13668.941} C_VEL
LIN {X 0,Y 347.444,Z 414.834,A -85,B 0,C 180,E1 -13670.687,E2 -13670.687} C_VEL
LIN {X 0,Y 346.989,Z 421.103,A -85,B 0,C 180,E1 -13672.435,E2 -13672.435} C_VEL
LIN {X 0,Y 346.735,Z 426.058,A -85,B 0,C 180,E1 -13674.183,E2 -13674.183} C_VEL
LIN {X 0,Y 346.562,Z 429.831,A -85,B 0,C 180,E1 -13675.93,E2 -13675.93} C_VEL
LIN {X 0,Y 346.495,Z 432.529,A -85,B 0,C 180,E1 -13677.675,E2 -13677.675} C_VEL
LIN {X 0,Y 346.455,Z 433.746,A -85,B 0,C 180,E1 -13678.838,E2 -13678.838} C_VEL
LIN {X 0,Y 346.435,Z 434.549,A -85,B 0,C 180,E1 -13680,E2 -13680} C_VEL
LIN {X 0,Y 346.488,Z 434.939,A -85,B 0,C 180,E1 -13681.162,E2 -13681.162} C_VEL
LIN {X 0,Y 346.627,Z 434.847,A -85,B 0,C 180,E1 -13682.324,E2 -13682.324} C_VEL
LIN {X 0,Y 346.827,Z 434.341,A -85,B 0,C 180,E1 -13683.485,E2 -13683.485} C_VEL
LIN {X 0,Y 347.064,Z 433.422,A -85,B 0,C 180,E1 -13684.646,E2 -13684.646} C_VEL
LIN {X 0,Y 347.201,Z 432.045,A -85,B 0,C 180,E1 -13685.809,E2 -13685.809} C_VEL
LIN {X 0,Y 347.534,Z 429.503,A -85,B 0,C 180,E1 -13687.375,E2 -13687.375} C_VEL
LIN {X 0,Y 348.394,Z 425.126,A -85,B 0,C 180,E1 -13689.287,E2 -13689.287} C_VEL
LIN {X 0,Y 349.095,Z 419.932,A -85,B 0,C 180,E1 -13691.026,E2 -13691.026} C_VEL
LIN {X 0,Y 350.155,Z 413.409,A -85,B 0,C 180,E1 -13692.755,E2 -13692.755} C_VEL
LIN {X 0,Y 351.442,Z 405.221,A -85,B 0,C 180,E1 -13694.476,E2 -13694.476} C_VEL
LIN {X 0,Y 352.707,Z 396.892,A -85,B 0,C 180,E1 -13695.901,E2 -13695.901} C_VEL
LIN {X 0,Y 354.093,Z 386.838,A -85,B 0,C 180,E1 -13697.321,E2 -13697.321} C_VEL
LIN {X 0,Y 355.46,Z 375.782,A -85,B 0,C 180,E1 -13698.591,E2 -13698.591} C_VEL
LIN {X 0,Y 356.841,Z 363.585,A -85,B 0,C 180,E1 -13699.693,E2 -13699.693} C_VEL
LIN {X 0,Y 357.111,Z 360.469,A -85,B 0,C 180,E1 -13699.941,E2 -13699.941} C_VEL
LIN {X 0,Y 354.752,Z 350.548,A -85,B 0,C 180,E1 -13700.958,E2 -13700.958} C_VEL
LIN {X 0,Y 351.12,Z 340.18,A -85,B 0,C 180,E1 -13702.013,E2 -13702.013} C_VEL
LIN {X 0,Y 348.677,Z 334.062,A -85,B 0,C 180,E1 -13702.635,E2 -13702.635} C_VEL
LIN {X 0,Y 348.988,Z 328.574,A -85,B 0,C 180,E1 -13706.298,E2 -13706.298} C_VEL
LIN {X 0,Y 349.569,Z 322.667,A -85,B 0,C 180,E1 -13710.173,E2 -13710.173} C_VEL
LIN {X 0,Y 350.031,Z 318.699,A -85,B 0,C 180,E1 -13712.828,E2 -13712.828} C_VEL
LIN {X 0,Y 349.981,Z 316.259,A -85,B 0,C 180,E1 -13714.581,E2 -13714.581} C_VEL
LIN {X 0,Y 349.414,Z 313.05,A -85,B 0,C 180,E1 -13717.115,E2 -13717.115} C_VEL
LIN {X 0,Y 348.625,Z 309.606,A -85,B 0,C 180,E1 -13720.173,E2 -13720.173} C_VEL
LIN {X 0,Y 347.974,Z 307.23,A -85,B 0,C 180,E1 -13722.824,E2 -13722.824} C_VEL
LIN {X 0,Y 349.273,Z 314.045,A -85,B 0,C 180,E1 -13726.418,E2 -13726.418} C_VEL
LIN {X 0,Y 350.704,Z 321.42,A -85,B 0,C 180,E1 -13730.113,E2 -13730.113} C_VEL
LIN {X 0,Y 351.506,Z 326.238,A -85,B 0,C 180,E1 -13732.424,E2 -13732.424} C_VEL
LIN {X 0,Y 351.413,Z 329.372,A -85,B 0,C 180,E1 -13733.844,E2 -13733.844} C_VEL
LIN {X 0,Y 350.371,Z 337.506,A -85,B 0,C 180,E1 -13737.402,E2 -13737.402} C_VEL
LIN {X 0,Y 349.541,Z 344.72,A -85,B 0,C 180,E1 -13740.488,E2 -13740.488} C_VEL
LIN {X 0,Y 348.667,Z 353.866,A -85,B 0,C 180,E1 -13744.318,E2 -13744.318} C_VEL
LIN {X 0,Y 347.881,Z 362.919,A -85,B 0,C 180,E1 -13748.053,E2 -13748.053} C_VEL
LIN {X 0,Y 348.704,Z 366.827,A -85,B 0,C 180,E1 -13748.31,E2 -13748.31} C_VEL
LIN {X 0,Y 351.08,Z 378.317,A -85,B 0,C 180,E1 -13749.11,E2 -13749.11} C_VEL
LIN {X 0,Y 352.251,Z 392.697,A -85,B 0,C 180,E1 -13750.173,E2 -13750.173} C_VEL
LIN {X 0,Y 353.076,Z 405.218,A -85,B 0,C 180,E1 -13751.314,E2 -13751.314} C_VEL
LIN {X 0,Y 352.724,Z 410.879,A -85,B 0,C 180,E1 -13751.861,E2 -13751.861} C_VEL
LIN {X 0,Y 351.284,Z 422.549,A -85,B 0,C 180,E1 -13753.136,E2 -13753.136} C_VEL
LIN {X 0,Y 349.988,Z 432.898,A -85,B 0,C 180,E1 -13754.553,E2 -13754.553} C_VEL
LIN {X 0,Y 348.976,Z 441.699,A -85,B 0,C 180,E1 -13756.015,E2 -13756.015} C_VEL
LIN {X 0,Y 347.945,Z 450.315,A -85,B 0,C 180,E1 -13757.755,E2 -13757.755} C_VEL
LIN {X 0,Y 347.155,Z 458.311,A -85,B 0,C 180,E1 -13759.797,E2 -13759.797} C_VEL
LIN {X 0,Y 346.638,Z 464.519,A -85,B 0,C 180,E1 -13761.841,E2 -13761.841} C_VEL
LIN {X 0,Y 346.402,Z 468.969,A -85,B 0,C 180,E1 -13763.795,E2 -13763.795} C_VEL
LIN {X 0,Y 346.324,Z 471.575,A -85,B 0,C 180,E1 -13765.344,E2 -13765.344} C_VEL
LIN {X 0,Y 346.297,Z 473.005,A -85,B 0,C 180,E1 -13766.509,E2 -13766.509} C_VEL
LIN {X 0,Y 346.304,Z 474.026,A -85,B 0,C 180,E1 -13767.674,E2 -13767.674} C_VEL
LIN {X 0,Y 346.467,Z 474.596,A -85,B 0,C 180,E1 -13768.838,E2 -13768.838} C_VEL
LIN {X 0,Y 346.467,Z 474.72,A -85,B 0,C 180,E1 -13770,E2 -13770} C_VEL
LIN {X 0,Y 346.465,Z 474.432,A -85,B 0,C 180,E1 -13771.162,E2 -13771.162} C_VEL
LIN {X 0,Y 346.338,Z 473.694,A -85,B 0,C 180,E1 -13772.326,E2 -13772.326} C_VEL
LIN {X 0,Y 346.347,Z 471.065,A -85,B 0,C 180,E1 -13774.656,E2 -13774.656} C_VEL
LIN {X 0,Y 346.448,Z 468.312,A -85,B 0,C 180,E1 -13776.274,E2 -13776.274} C_VEL
LIN {X 0,Y 346.616,Z 463.955,A -85,B 0,C 180,E1 -13778.16,E2 -13778.16} C_VEL
LIN {X 0,Y 347.14,Z 457.654,A -85,B 0,C 180,E1 -13780.204,E2 -13780.204} C_VEL
LIN {X 0,Y 347.783,Z 450.782,A -85,B 0,C 180,E1 -13781.954,E2 -13781.954} C_VEL
LIN {X 0,Y 349.148,Z 439.352,A -85,B 0,C 180,E1 -13784.275,E2 -13784.275} C_VEL
LIN {X 0,Y 350.399,Z 428.827,A -85,B 0,C 180,E1 -13786.009,E2 -13786.009} C_VEL
LIN {X 0,Y 351.866,Z 418.189,A -85,B 0,C 180,E1 -13787.434,E2 -13787.434} C_VEL
LIN {X 0,Y 353.259,Z 406.481,A -85,B 0,C 180,E1 -13788.712,E2 -13788.712} C_VEL
LIN {X 0,Y 352.843,Z 394.229,A -85,B 0,C 180,E1 -13789.921,E2 -13789.921} C_VEL
LIN {X 0,Y 352.155,Z 382.178,A -85,B 0,C 180,E1 -13790.927,E2 -13790.927} C_VEL
LIN {X 0,Y 350.169,Z 369.826,A -85,B 0,C 180,E1 -13791.884,E2 -13791.884} C_VEL
LIN {X 0,Y 347.889,Z 359.686,A -85,B 0,C 180,E1 -13792.65,E2 -13792.65} C_VEL
LIN {X 0,Y 348.656,Z 351.072,A -85,B 0,C 180,E1 -13796.325,E2 -13796.325} C_VEL
LIN {X 0,Y 349.638,Z 342.548,A -85,B 0,C 180,E1 -13800.193,E2 -13800.193} C_VEL
LIN {X 0,Y 350.655,Z 335.911,A -85,B 0,C 180,E1 -13803.447,E2 -13803.447} C_VEL
LIN {X 0,Y 351.881,Z 329.683,A -85,B 0,C 180,E1 -13806.811,E2 -13806.811} C_VEL
LIN {X 0,Y 351.705,Z 326.587,A -85,B 0,C 180,E1 -13808.801,E2 -13808.801} C_VEL
LIN {X 0,Y 350.88,Z 322.245,A -85,B 0,C 180,E1 -13812.175,E2 -13812.175} C_VEL
LIN {X 0,Y 350.279,Z 318.99,A -85,B 0,C 180,E1 -13815.393,E2 -13815.393} C_VEL
LIN {X 0,Y 349.871,Z 316.696,A -85,B 0,C 180,E1 -13818.48,E2 -13818.48} C_VEL
LIN {X 0,Y 349.558,Z 315.163,A -85,B 0,C 180,E1 -13821.639,E2 -13821.639} C_VEL
LIN {X 0,Y 349.348,Z 314.458,A -85,B 0,C 180,E1 -13824.309,E2 -13824.309} C_VEL
LIN {X 0,Y 349.247,Z 314.221,A -85,B 0,C 180,E1 -13827.691,E2 -13827.691} C_VEL
LIN {X 0,Y 349.278,Z 314.617,A -85,B 0,C 180,E1 -13831.124,E2 -13831.124} C_VEL
LIN {X 0,Y 349.309,Z 315.292,A -85,B 0,C 180,E1 -13833.728,E2 -13833.728} C_VEL
LIN {X 0,Y 349.186,Z 316.501,A -85,B 0,C 180,E1 -13836.892,E2 -13836.892} C_VEL
LIN {X 0,Y 349.167,Z 316.893,A -85,B 0,C 180,E1 -13837.496,E2 -13837.496} C_VEL
LIN {X 0,Y 350.484,Z 319.821,A -85,B 0,C 180,E1 -13837.823,E2 -13837.823} C_VEL
LIN {X 0,Y 354.958,Z 329.331,A -85,B 0,C 180,E1 -13838.97,E2 -13838.97} C_VEL
LIN {X 0,Y 357.941,Z 337.963,A -85,B 0,C 180,E1 -13839.971,E2 -13839.971} C_VEL
LIN {X 0,Y 358.169,Z 339.349,A -85,B 0,C 180,E1 -13840.117,E2 -13840.117} C_VEL
LIN {X 0,Y 356.848,Z 351.966,A -85,B 0,C 180,E1 -13841.236,E2 -13841.236} C_VEL
LIN {X 0,Y 355.495,Z 362.882,A -85,B 0,C 180,E1 -13842.453,E2 -13842.453} C_VEL
LIN {X 0,Y 354.351,Z 371.215,A -85,B 0,C 180,E1 -13843.583,E2 -13843.583} C_VEL
LIN {X 0,Y 353.001,Z 379.982,A -85,B 0,C 180,E1 -13845,E2 -13845} C_VEL
LIN {X 0,Y 351.669,Z 388.517,A -85,B 0,C 180,E1 -13846.713,E2 -13846.713} C_VEL
LIN {X 0,Y 350.423,Z 395.405,A -85,B 0,C 180,E1 -13848.43,E2 -13848.43} C_VEL
LIN {X 0,Y 349.579,Z 400.685,A -85,B 0,C 180,E1 -13850.1,E2 -13850.1} C_VEL
LIN {X 0,Y 348.649,Z 405.143,A -85,B 0,C 180,E1 -13851.888,E2 -13851.888} C_VEL
LIN {X 0,Y 348.254,Z 407.33,A -85,B 0,C 180,E1 -13853.045,E2 -13853.045} C_VEL
LIN {X 0,Y 347.941,Z 409.072,A -85,B 0,C 180,E1 -13854.204,E2 -13854.204} C_VEL
LIN {X 0,Y 347.588,Z 410.398,A -85,B 0,C 180,E1 -13855.361,E2 -13855.361} C_VEL
LIN {X 0,Y 347.219,Z 411.261,A -85,B 0,C 180,E1 -13856.519,E2 -13856.519} C_VEL
LIN {X 0,Y 346.949,Z 411.712,A -85,B 0,C 180,E1 -13857.678,E2 -13857.678} C_VEL
LIN {X 0,Y 346.803,Z 411.751,A -85,B 0,C 180,E1 -13858.839,E2 -13858.839} C_VEL
LIN {X 0,Y 346.75,Z 411.338,A -85,B 0,C 180,E1 -13860,E2 -13860} C_VEL
LIN {X 0,Y 346.783,Z 410.486,A -85,B 0,C 180,E1 -13861.161,E2 -13861.161} C_VEL
LIN {X 0,Y 346.845,Z 409.224,A -85,B 0,C 180,E1 -13862.323,E2 -13862.323} C_VEL
LIN {X 0,Y 347.088,Z 406.493,A -85,B 0,C 180,E1 -13864.064,E2 -13864.064} C_VEL
LIN {X 0,Y 347.238,Z 402.731,A -85,B 0,C 180,E1 -13865.808,E2 -13865.808} C_VEL
LIN {X 0,Y 347.552,Z 397.176,A -85,B 0,C 180,E1 -13867.755,E2 -13867.755} C_VEL
LIN {X 0,Y 348.019,Z 390.421,A -85,B 0,C 180,E1 -13869.59,E2 -13869.59} C_VEL
LIN {X 0,Y 348.63,Z 382.443,A -85,B 0,C 180,E1 -13871.335,E2 -13871.335} C_VEL
LIN {X 0,Y 349.232,Z 374.333,A -85,B 0,C 180,E1 -13872.789,E2 -13872.789} C_VEL
LIN {X 0,Y 350.13,Z 363.409,A -85,B 0,C 180,E1 -13874.383,E2 -13874.383} C_VEL
LIN {X 0,Y 350.891,Z 352.292,A -85,B 0,C 180,E1 -13875.7,E2 -13875.7} C_VEL
LIN {X 0,Y 351.601,Z 340.156,A -85,B 0,C 180,E1 -13876.848,E2 -13876.848} C_VEL
LIN {X 0,Y 352.274,Z 328.809,A -85,B 0,C 180,E1 -13877.7,E2 -13877.7} C_VEL
LIN {X 0,Y 349.812,Z 317.243,A -85,B 0,C 180,E1 -13878.492,E2 -13878.492} C_VEL
LIN {X 0,Y 347.179,Z 306.263,A -85,B 0,C 180,E1 -13879.09,E2 -13879.09} C_VEL
LIN {X 0,Y 347.476,Z 306.201,A -85,B 0,C 180,E1 -13882.6,E2 -13882.6} C_VEL
LIN {X 0,Y 347.692,Z 306.171,A -85,B 0,C 180,E1 -13885.118,E2 -13885.118} C_VEL
LIN {X 0,Y 347.762,Z 306.161,A -85,B 0,C 180,E1 -13887.698,E2 -13887.698} C_VEL
LIN {X 0,Y 347.751,Z 306.165,A -85,B 0,C 180,E1 -13890.348,E2 -13890.348} C_VEL
LIN {X 0,Y 347.75,Z 306.17,A -85,B 0,C 180,E1 -13894.044,E2 -13894.044} C_VEL
LIN {X 0,Y 347.764,Z 306.168,A -85,B 0,C 180,E1 -13897.321,E2 -13897.321} C_VEL
LIN {X 0,Y 347.735,Z 306.175,A -85,B 0,C 180,E1 -13900.297,E2 -13900.297} C_VEL
LIN {X 0,Y 347.725,Z 306.173,A -85,B 0,C 180,E1 -13903.408,E2 -13903.408} C_VEL
LIN {X 0,Y 347.727,Z 306.168,A -85,B 0,C 180,E1 -13906.686,E2 -13906.686} C_VEL
LIN {X 0,Y 347.75,Z 306.169,A -85,B 0,C 180,E1 -13910.173,E2 -13910.173} C_VEL
LIN {X 0,Y 347.752,Z 306.167,A -85,B 0,C 180,E1 -13912.678,E2 -13912.678} C_VEL
LIN {X 0,Y 347.729,Z 306.295,A -85,B 0,C 180,E1 -13915.446,E2 -13915.446} C_VEL
LIN {X 0,Y 347.58,Z 310.613,A -85,B 0,C 180,E1 -13918.283,E2 -13918.283} C_VEL
LIN {X 0,Y 347.405,Z 316.755,A -85,B 0,C 180,E1 -13922.271,E2 -13922.271} C_VEL
LIN {X 0,Y 347.297,Z 322.951,A -85,B 0,C 180,E1 -13926.126,E2 -13926.126} C_VEL
LIN {X 0,Y 347.37,Z 328.397,A -85,B 0,C 180,E1 -13929.208,E2 -13929.208} C_VEL
LIN {X 0,Y 351.181,Z 341.909,A -85,B 0,C 180,E1 -13929.941,E2 -13929.941} C_VEL
LIN {X 0,Y 353.848,Z 353.752,A -85,B 0,C 180,E1 -13930.761,E2 -13930.761} C_VEL
LIN {X 0,Y 354.576,Z 358.011,A -85,B 0,C 180,E1 -13931.101,E2 -13931.101} C_VEL
LIN {X 0,Y 353.61,Z 370.113,A -85,B 0,C 180,E1 -13932.057,E2 -13932.057} C_VEL
LIN {X 0,Y 352.534,Z 381.15,A -85,B 0,C 180,E1 -13933.188,E2 -13933.188} C_VEL
LIN {X 0,Y 351.604,Z 391.273,A -85,B 0,C 180,E1 -13934.494,E2 -13934.494} C_VEL
LIN {X 0,Y 350.593,Z 399.514,A -85,B 0,C 180,E1 -13935.785,E2 -13935.785} C_VEL
LIN {X 0,Y 349.444,Z 408.439,A -85,B 0,C 180,E1 -13937.514,E2 -13937.514} C_VEL
LIN {X 0,Y 348.524,Z 415.603,A -85,B 0,C 180,E1 -13939.25,E2 -13939.25} C_VEL
LIN {X 0,Y 347.693,Z 422.165,A -85,B 0,C 180,E1 -13941.28,E2 -13941.28} C_VEL
LIN {X 0,Y 347.216,Z 426.472,A -85,B 0,C 180,E1 -13943.024,E2 -13943.024} C_VEL
LIN {X 0,Y 346.892,Z 428.744,A -85,B 0,C 180,E1 -13944.186,E2 -13944.186} C_VEL
LIN {X 0,Y 346.702,Z 430.592,A -85,B 0,C 180,E1 -13945.349,E2 -13945.349} C_VEL
LIN {X 0,Y 346.676,Z 431.994,A -85,B 0,C 180,E1 -13946.513,E2 -13946.513} C_VEL
LIN {X 0,Y 346.573,Z 432.983,A -85,B 0,C 180,E1 -13947.676,E2 -13947.676} C_VEL
LIN {X 0,Y 346.408,Z 433.831,A -85,B 0,C 180,E1 -13950,E2 -13950} C_VEL
LIN {X 0,Y 346.571,Z 433.051,A -85,B 0,C 180,E1 -13952.324,E2 -13952.324} C_VEL
LIN {X 0,Y 346.654,Z 432.09,A -85,B 0,C 180,E1 -13953.487,E2 -13953.487} C_VEL
LIN {X 0,Y 346.678,Z 430.741,A -85,B 0,C 180,E1 -13954.651,E2 -13954.651} C_VEL
LIN {X 0,Y 347.064,Z 427.882,A -85,B 0,C 180,E1 -13956.395,E2 -13956.395} C_VEL
LIN {X 0,Y 347.467,Z 424.005,A -85,B 0,C 180,E1 -13958.14,E2 -13958.14} C_VEL
LIN {X 0,Y 348.047,Z 418.98,A -85,B 0,C 180,E1 -13959.883,E2 -13959.883} C_VEL
LIN {X 0,Y 348.96,Z 412.626,A -85,B 0,C 180,E1 -13961.619,E2 -13961.619} C_VEL
LIN {X 0,Y 349.973,Z 404.732,A -85,B 0,C 180,E1 -13963.352,E2 -13963.352} C_VEL
LIN {X 0,Y 351.006,Z 396.659,A -85,B 0,C 180,E1 -13964.791,E2 -13964.791} C_VEL
LIN {X 0,Y 352.093,Z 386.745,A -85,B 0,C 180,E1 -13966.227,E2 -13966.227} C_VEL
LIN {X 0,Y 352.984,Z 376.95,A -85,B 0,C 180,E1 -13967.377,E2 -13967.377} C_VEL
LIN {X 0,Y 354.026,Z 366.306,A -85,B 0,C 180,E1 -13968.37,E2 -13968.37} C_VEL
LIN {X 0,Y 354.574,Z 357.369,A -85,B 0,C 180,E1 -13969.049,E2 -13969.049} C_VEL
LIN {X 0,Y 351.874,Z 344.548,A -85,B 0,C 180,E1 -13969.995,E2 -13969.995} C_VEL
LIN {X 0,Y 348.315,Z 331.731,A -85,B 0,C 180,E1 -13970.74,E2 -13970.74} C_VEL
LIN {X 0,Y 347.367,Z 328.185,A -85,B 0,C 180,E1 -13970.923,E2 -13970.923} C_VEL
LIN {X 0,Y 347.319,Z 322.246,A -85,B 0,C 180,E1 -13974.414,E2 -13974.414} C_VEL
LIN {X 0,Y 347.426,Z 315.929,A -85,B 0,C 180,E1 -13978.384,E2 -13978.384} C_VEL
LIN {X 0,Y 347.592,Z 310.572,A -85,B 0,C 180,E1 -13981.874,E2 -13981.874} C_VEL
LIN {X 0,Y 347.743,Z 306.314,A -85,B 0,C 180,E1 -13984.64,E2 -13984.64} C_VEL
LIN {X 0,Y 347.758,Z 306.167,A -85,B 0,C 180,E1 -13988.259,E2 -13988.259} C_VEL
LIN {X 0,Y 347.071,Z 306.254,A -85,B 0,C 180,E1 -13989.226,E2 -13989.226} C_VEL
LIN {X 0,Y 344.205,Z 306.613,A -85,B 0,C 180,E1 -13990.799,E2 -13990.799} C_VEL
LIN {X 0,Y 341.785,Z 306.914,A -85,B 0,C 180,E1 -13992.072,E2 -13992.072} C_VEL
LIN {X 0,Y 340.743,Z 307.045,A -85,B 0,C 180,E1 -13993.057,E2 -13993.057} C_VEL
LIN {X 0,Y 340.655,Z 307.053,A -85,B 0,C 180,E1 -13993.39,E2 -13993.39} C_VEL
LIN {X 0,Y 340.678,Z 307.051,A -85,B 0,C 180,E1 -13997.096,E2 -13997.096} C_VEL
LIN {X 0,Y 340.701,Z 307.048,A -85,B 0,C 180,E1 -14000.247,E2 -14000.247} C_VEL
LIN {X 0,Y 340.666,Z 307.051,A -85,B 0,C 180,E1 -14003.57,E2 -14003.57} C_VEL
LIN {X 0,Y 340.474,Z 307.194,A -85,B 0,C 180,E1 -14007.014,E2 -14007.014} C_VEL
LIN {X 0,Y 340.103,Z 314.353,A -85,B 0,C 180,E1 -14011.622,E2 -14011.622} C_VEL
LIN {X 0,Y 340.01,Z 320.296,A -85,B 0,C 180,E1 -14015.434,E2 -14015.434} C_VEL
LIN {X 0,Y 339.922,Z 325.121,A -85,B 0,C 180,E1 -14018.496,E2 -14018.496} C_VEL
LIN {X 0,Y 339.874,Z 328.616,A -85,B 0,C 180,E1 -14020.72,E2 -14020.72} C_VEL
LIN {X 0,Y 342.742,Z 343.138,A -85,B 0,C 180,E1 -14021.509,E2 -14021.509} C_VEL
LIN {X 0,Y 344.767,Z 354.044,A -85,B 0,C 180,E1 -14022.272,E2 -14022.272} C_VEL
LIN {X 0,Y 344.131,Z 366.294,A -85,B 0,C 180,E1 -14023.234,E2 -14023.234} C_VEL
LIN {X 0,Y 343.297,Z 378.37,A -85,B 0,C 180,E1 -14024.444,E2 -14024.444} C_VEL
LIN {X 0,Y 342.524,Z 388.908,A -85,B 0,C 180,E1 -14025.746,E2 -14025.746} C_VEL
LIN {X 0,Y 341.658,Z 398.651,A -85,B 0,C 180,E1 -14027.224,E2 -14027.224} C_VEL
LIN {X 0,Y 340.951,Z 408.191,A -85,B 0,C 180,E1 -14029.008,E2 -14029.008} C_VEL
LIN {X 0,Y 340.331,Z 415.825,A -85,B 0,C 180,E1 -14030.791,E2 -14030.791} C_VEL
LIN {X 0,Y 339.831,Z 422.893,A -85,B 0,C 180,E1 -14032.872,E2 -14032.872} C_VEL
LIN {X 0,Y 339.613,Z 427.532,A -85,B 0,C 180,E1 -14034.657,E2 -14034.657} C_VEL
LIN {X 0,Y 339.457,Z 431.036,A -85,B 0,C 180,E1 -14036.439,E2 -14036.439} C_VEL
LIN {X 0,Y 339.404,Z 432.801,A -85,B 0,C 180,E1 -14037.626,E2 -14037.626} C_VEL
LIN {X 0,Y 339.375,Z 434.104,A -85,B 0,C 180,E1 -14038.813,E2 -14038.813} C_VEL
LIN {X 0,Y 339.372,Z 434.954,A -85,B 0,C 180,E1 -14040,E2 -14040} C_VEL
LIN {X 0,Y 339.427,Z 435.395,A -85,B 0,C 180,E1 -14041.186,E2 -14041.186} C_VEL
LIN {X 0,Y 339.573,Z 435.384,A -85,B 0,C 180,E1 -14042.372,E2 -14042.372} C_VEL
LIN {X 0,Y 339.784,Z 434.926,A -85,B 0,C 180,E1 -14043.558,E2 -14043.558} C_VEL
LIN {X 0,Y 340.032,Z 434.067,A -85,B 0,C 180,E1 -14044.742,E2 -14044.742} C_VEL
LIN {X 0,Y 340.175,Z 432.768,A -85,B 0,C 180,E1 -14045.929,E2 -14045.929} C_VEL
LIN {X 0,Y 340.509,Z 430.438,A -85,B 0,C 180,E1 -14047.455,E2 -14047.455} C_VEL
LIN {X 0,Y 341.458,Z 426.037,A -85,B 0,C 180,E1 -14049.477,E2 -14049.477} C_VEL
LIN {X 0,Y 342.235,Z 420.988,A -85,B 0,C 180,E1 -14051.25,E2 -14051.25} C_VEL
LIN {X 0,Y 343.344,Z 414.591,A -85,B 0,C 180,E1 -14053.012,E2 -14053.012} C_VEL
LIN {X 0,Y 344.721,Z 406.582,A -85,B 0,C 180,E1 -14054.764,E2 -14054.764} C_VEL
LIN {X 0,Y 346.034,Z 398.498,A -85,B 0,C 180,E1 -14056.216,E2 -14056.216} C_VEL
LIN {X 0,Y 347.532,Z 388.725,A -85,B 0,C 180,E1 -14057.658,E2 -14057.658} C_VEL
LIN {X 0,Y 349.14,Z 376.659,A -85,B 0,C 180,E1 -14059.093,E2 -14059.093} C_VEL
LIN {X 0,Y 350.669,Z 364.196,A -85,B 0,C 180,E1 -14060.257,E2 -14060.257} C_VEL
LIN {X 0,Y 350.868,Z 362.33,A -85,B 0,C 180,E1 -14060.414,E2 -14060.414} C_VEL
LIN {X 0,Y 348.45,Z 352.137,A -85,B 0,C 180,E1 -14061.518,E2 -14061.518} C_VEL
LIN {X 0,Y 344.627,Z 341.329,A -85,B 0,C 180,E1 -14062.703,E2 -14062.703} C_VEL
LIN {X 0,Y 341.907,Z 334.728,A -85,B 0,C 180,E1 -14063.469,E2 -14063.469} C_VEL
LIN {X 0,Y 342.213,Z 329.746,A -85,B 0,C 180,E1 -14066.86,E2 -14066.86} C_VEL
LIN {X 0,Y 342.847,Z 324.324,A -85,B 0,C 180,E1 -14070.575,E2 -14070.575} C_VEL
LIN {X 0,Y 343.343,Z 320.098,A -85,B 0,C 180,E1 -14073.551,E2 -14073.551} C_VEL
LIN {X 0,Y 343.254,Z 318.203,A -85,B 0,C 180,E1 -14075.016,E2 -14075.016} C_VEL
LIN {X 0,Y 342.673,Z 314.772,A -85,B 0,C 180,E1 -14077.972,E2 -14077.972} C_VEL
LIN {X 0,Y 341.939,Z 311.677,A -85,B 0,C 180,E1 -14081.125,E2 -14081.125} C_VEL
LIN {X 0,Y 341.408,Z 310.223,A -85,B 0,C 180,E1 -14083.044,E2 -14083.044} C_VEL
LIN {X 0,Y 341.263,Z 310.023,A -85,B 0,C 180,E1 -14083.52,E2 -14083.52} C_VEL
LIN {X 0,Y 342.418,Z 315.945,A -85,B 0,C 180,E1 -14086.678,E2 -14086.678} C_VEL
LIN {X 0,Y 343.669,Z 322.396,A -85,B 0,C 180,E1 -14089.967,E2 -14089.967} C_VEL
LIN {X 0,Y 344.483,Z 327.078,A -85,B 0,C 180,E1 -14092.262,E2 -14092.262} C_VEL
LIN {X 0,Y 344.412,Z 330.216,A -85,B 0,C 180,E1 -14093.717,E2 -14093.717} C_VEL
LIN {X 0,Y 343.428,Z 337.648,A -85,B 0,C 180,E1 -14097.039,E2 -14097.039} C_VEL
LIN {X 0,Y 342.46,Z 345.543,A -85,B 0,C 180,E1 -14100.493,E2 -14100.493} C_VEL
LIN {X 0,Y 341.563,Z 354.663,A -85,B 0,C 180,E1 -14104.399,E2 -14104.399} C_VEL
LIN {X 0,Y 340.969,Z 361.305,A -85,B 0,C 180,E1 -14107.208,E2 -14107.208} C_VEL
LIN {X 0,Y 341.777,Z 365.364,A -85,B 0,C 180,E1 -14107.5,E2 -14107.5} C_VEL
LIN {X 0,Y 344.525,Z 377.99,A -85,B 0,C 180,E1 -14108.458,E2 -14108.458} C_VEL
LIN {X 0,Y 345.626,Z 391.004,A -85,B 0,C 180,E1 -14109.469,E2 -14109.469} C_VEL
LIN {X 0,Y 346.316,Z 403.928,A -85,B 0,C 180,E1 -14110.665,E2 -14110.665} C_VEL
LIN {X 0,Y 346.427,Z 409.135,A -85,B 0,C 180,E1 -14111.213,E2 -14111.213} C_VEL
LIN {X 0,Y 344.844,Z 420.919,A -85,B 0,C 180,E1 -14112.506,E2 -14112.506} C_VEL
LIN {X 0,Y 343.351,Z 431.926,A -85,B 0,C 180,E1 -14114.02,E2 -14114.02} C_VEL
LIN {X 0,Y 342.092,Z 441.946,A -85,B 0,C 180,E1 -14115.728,E2 -14115.728} C_VEL
LIN {X 0,Y 340.992,Z 450.37,A -85,B 0,C 180,E1 -14117.502,E2 -14117.502} C_VEL
LIN {X 0,Y 340.246,Z 457.226,A -85,B 0,C 180,E1 -14119.286,E2 -14119.286} C_VEL
LIN {X 0,Y 339.704,Z 462.763,A -85,B 0,C 180,E1 -14121.074,E2 -14121.074} C_VEL
LIN {X 0,Y 339.436,Z 467.131,A -85,B 0,C 180,E1 -14122.864,E2 -14122.864} C_VEL
LIN {X 0,Y 339.298,Z 469.449,A -85,B 0,C 180,E1 -14124.055,E2 -14124.055} C_VEL
LIN {X 0,Y 339.242,Z 471.272,A -85,B 0,C 180,E1 -14125.247,E2 -14125.247} C_VEL
LIN {X 0,Y 339.215,Z 472.679,A -85,B 0,C 180,E1 -14126.436,E2 -14126.436} C_VEL
LIN {X 0,Y 339.208,Z 473.667,A -85,B 0,C 180,E1 -14127.625,E2 -14127.625} C_VEL
LIN {X 0,Y 339.379,Z 474.193,A -85,B 0,C 180,E1 -14128.813,E2 -14128.813} C_VEL
LIN {X 0,Y 339.402,Z 474.295,A -85,B 0,C 180,E1 -14130,E2 -14130} C_VEL
LIN {X 0,Y 339.397,Z 473.984,A -85,B 0,C 180,E1 -14131.187,E2 -14131.187} C_VEL
LIN {X 0,Y 339.21,Z 472.106,A -85,B 0,C 180,E1 -14133.564,E2 -14133.564} C_VEL
LIN {X 0,Y 339.262,Z 470.648,A -85,B 0,C 180,E1 -14134.753,E2 -14134.753} C_VEL
LIN {X 0,Y 339.344,Z 468.227,A -85,B 0,C 180,E1 -14136.222,E2 -14136.222} C_VEL
LIN {X 0,Y 339.565,Z 463.538,A -85,B 0,C 180,E1 -14138.33,E2 -14138.33} C_VEL
LIN {X 0,Y 340.101,Z 457.236,A -85,B 0,C 180,E1 -14140.417,E2 -14140.417} C_VEL
LIN {X 0,Y 340.812,Z 450.367,A -85,B 0,C 180,E1 -14142.203,E2 -14142.203} C_VEL
LIN {X 0,Y 342.007,Z 440.77,A -85,B 0,C 180,E1 -14144.276,E2 -14144.276} C_VEL
LIN {X 0,Y 343.288,Z 430.864,A -85,B 0,C 180,E1 -14146.044,E2 -14146.044} C_VEL
LIN {X 0,Y 344.939,Z 419.683,A -85,B 0,C 180,E1 -14147.642,E2 -14147.642} C_VEL
LIN {X 0,Y 346.54,Z 408.618,A -85,B 0,C 180,E1 -14148.935,E2 -14148.935} C_VEL
LIN {X 0,Y 346.288,Z 395.546,A -85,B 0,C 180,E1 -14150.314,E2 -14150.314} C_VEL
LIN {X 0,Y 345.799,Z 384.099,A -85,B 0,C 180,E1 -14151.335,E2 -14151.335} C_VEL
LIN {X 0,Y 344.012,Z 371.91,A -85,B 0,C 180,E1 -14152.363,E2 -14152.363} C_VEL
LIN {X 0,Y 341.563,Z 361.62,A -85,B 0,C 180,E1 -14153.211,E2 -14153.211} C_VEL
LIN {X 0,Y 340.98,Z 358.661,A -85,B 0,C 180,E1 -14153.457,E2 -14153.457} C_VEL
LIN {X 0,Y 341.724,Z 350.873,A -85,B 0,C 180,E1 -14156.902,E2 -14156.902} C_VEL
LIN {X 0,Y 342.843,Z 342.54,A -85,B 0,C 180,E1 -14160.829,E2 -14160.829} C_VEL
LIN {X 0,Y 343.923,Z 335.989,A -85,B 0,C 180,E1 -14164.191,E2 -14164.191} C_VEL
LIN {X 0,Y 344.728,Z 332.29,A -85,B 0,C 180,E1 -14166.244,E2 -14166.244} C_VEL
LIN {X 0,Y 345.006,Z 329.945,A -85,B 0,C 180,E1 -14167.671,E2 -14167.671} C_VEL
LIN {X 0,Y 344.544,Z 326.704,A -85,B 0,C 180,E1 -14169.981,E2 -14169.981} C_VEL
LIN {X 0,Y 343.932,Z 323.543,A -85,B 0,C 180,E1 -14172.639,E2 -14172.639} C_VEL
LIN {X 0,Y 343.347,Z 320.442,A -85,B 0,C 180,E1 -14175.897,E2 -14175.897} C_VEL
LIN {X 0,Y 342.916,Z 318.115,A -85,B 0,C 180,E1 -14179.316,E2 -14179.316} C_VEL
LIN {X 0,Y 342.678,Z 316.907,A -85,B 0,C 180,E1 -14182.028,E2 -14182.028} C_VEL
LIN {X 0,Y 342.457,Z 316.167,A -85,B 0,C 180,E1 -14185.174,E2 -14185.174} C_VEL
LIN {X 0,Y 342.393,Z 316.002,A -85,B 0,C 180,E1 -14187.746,E2 -14187.746} C_VEL
LIN {X 0,Y 342.402,Z 316.469,A -85,B 0,C 180,E1 -14191.83,E2 -14191.83} C_VEL
LIN {X 0,Y 342.383,Z 317.22,A -85,B 0,C 180,E1 -14194.579,E2 -14194.579} C_VEL
LIN {X 0,Y 342.309,Z 318.079,A -85,B 0,C 180,E1 -14196.68,E2 -14196.68} C_VEL
LIN {X 0,Y 343.614,Z 320.99,A -85,B 0,C 180,E1 -14197.035,E2 -14197.035} C_VEL
LIN {X 0,Y 348.118,Z 330.003,A -85,B 0,C 180,E1 -14198.23,E2 -14198.23} C_VEL
LIN {X 0,Y 351.562,Z 339.728,A -85,B 0,C 180,E1 -14199.443,E2 -14199.443} C_VEL
LIN {X 0,Y 351.959,Z 341.612,A -85,B 0,C 180,E1 -14199.657,E2 -14199.657} C_VEL
LIN {X 0,Y 350.658,Z 352.93,A -85,B 0,C 180,E1 -14200.701,E2 -14200.701} C_VEL
LIN {X 0,Y 349.134,Z 363.989,A -85,B 0,C 180,E1 -14201.971,E2 -14201.971} C_VEL
LIN {X 0,Y 347.794,Z 373.245,A -85,B 0,C 180,E1 -14203.264,E2 -14203.264} C_VEL
LIN {X 0,Y 346.353,Z 381.748,A -85,B 0,C 180,E1 -14204.705,E2 -14204.705} C_VEL
LIN {X 0,Y 344.946,Z 390.033,A -85,B 0,C 180,E1 -14206.449,E2 -14206.449} C_VEL
LIN {X 0,Y 343.608,Z 396.808,A -85,B 0,C 180,E1 -14208.198,E2 -14208.198} C_VEL
LIN {X 0,Y 342.53,Z 402.623,A -85,B 0,C 180,E1 -14210.157,E2 -14210.157} C_VEL
LIN {X 0,Y 341.501,Z 407.369,A -85,B 0,C 180,E1 -14212.313,E2 -14212.313} C_VEL
LIN {X 0,Y 340.947,Z 410.064,A -85,B 0,C 180,E1 -14214.084,E2 -14214.084} C_VEL
LIN {X 0,Y 340.575,Z 411.311,A -85,B 0,C 180,E1 -14215.265,E2 -14215.265} C_VEL
LIN {X 0,Y 340.193,Z 412.118,A -85,B 0,C 180,E1 -14216.447,E2 -14216.447} C_VEL
LIN {X 0,Y 339.912,Z 412.513,A -85,B 0,C 180,E1 -14217.63,E2 -14217.63} C_VEL
LIN {X 0,Y 339.758,Z 412.486,A -85,B 0,C 180,E1 -14218.815,E2 -14218.815} C_VEL
LIN {X 0,Y 339.702,Z 411.992,A -85,B 0,C 180,E1 -14220,E2 -14220} C_VEL
LIN {X 0,Y 339.738,Z 411.086,A -85,B 0,C 180,E1 -14221.185,E2 -14221.185} C_VEL
LIN {X 0,Y 339.779,Z 409.776,A -85,B 0,C 180,E1 -14222.371,E2 -14222.371} C_VEL
LIN {X 0,Y 340.04,Z 406.94,A -85,B 0,C 180,E1 -14224.148,E2 -14224.148} C_VEL
LIN {X 0,Y 340.175,Z 403.066,A -85,B 0,C 180,E1 -14225.929,E2 -14225.929} C_VEL
LIN {X 0,Y 340.468,Z 397.846,A -85,B 0,C 180,E1 -14227.765,E2 -14227.765} C_VEL
LIN {X 0,Y 340.982,Z 390.472,A -85,B 0,C 180,E1 -14229.79,E2 -14229.79} C_VEL
LIN {X 0,Y 341.643,Z 382.339,A -85,B 0,C 180,E1 -14231.57,E2 -14231.57} C_VEL
LIN {X 0,Y 342.473,Z 372.221,A -85,B 0,C 180,E1 -14233.348,E2 -14233.348} C_VEL
LIN {X 0,Y 343.341,Z 361.841,A -85,B 0,C 180,E1 -14234.825,E2 -14234.825} C_VEL
LIN {X 0,Y 344.094,Z 350.02,A -85,B 0,C 180,E1 -14236.183,E2 -14236.183} C_VEL
LIN {X 0,Y 344.841,Z 337.292,A -85,B 0,C 180,E1 -14237.341,E2 -14237.341} C_VEL
LIN {X 0,Y 345.299,Z 329.311,A -85,B 0,C 180,E1 -14237.931,E2 -14237.931} C_VEL
LIN {X 0,Y 342.326,Z 315.894,A -85,B 0,C 180,E1 -14238.855,E2 -14238.855} C_VEL
LIN {X 0,Y 340.142,Z 307.118,A -85,B 0,C 180,E1 -14239.344,E2 -14239.344} C_VEL
LIN {X 0,Y 340.487,Z 307.073,A -85,B 0,C 180,E1 -14243.09,E2 -14243.09} C_VEL
LIN {X 0,Y 340.653,Z 307.046,A -85,B 0,C 180,E1 -14245.674,E2 -14245.674} C_VEL
LIN {X 0,Y 340.707,Z 307.043,A -85,B 0,C 180,E1 -14248.323,E2 -14248.323} C_VEL
LIN {X 0,Y 340.7,Z 307.038,A -85,B 0,C 180,E1 -14251.045,E2 -14251.045} C_VEL
LIN {X 0,Y 340.72,Z 307.036,A -85,B 0,C 180,E1 -14255.279,E2 -14255.279} C_VEL
LIN {X 0,Y 340.712,Z 307.044,A -85,B 0,C 180,E1 -14258.386,E2 -14258.386} C_VEL
LIN {X 0,Y 340.701,Z 307.047,A -85,B 0,C 180,E1 -14262.046,E2 -14262.046} C_VEL
LIN {X 0,Y 340.654,Z 307.051,A -85,B 0,C 180,E1 -14266.227,E2 -14266.227} C_VEL
LIN {X 0,Y 340.691,Z 307.049,A -85,B 0,C 180,E1 -14269.753,E2 -14269.753} C_VEL
LIN {X 0,Y 340.687,Z 307.05,A -85,B 0,C 180,E1 -14273.256,E2 -14273.256} C_VEL
LIN {X 0,Y 340.684,Z 307.166,A -85,B 0,C 180,E1 -14275.208,E2 -14275.208} C_VEL
LIN {X 0,Y 340.627,Z 310.7,A -85,B 0,C 180,E1 -14277.558,E2 -14277.558} C_VEL
LIN {X 0,Y 340.431,Z 316.948,A -85,B 0,C 180,E1 -14281.652,E2 -14281.652} C_VEL
LIN {X 0,Y 340.319,Z 323.245,A -85,B 0,C 180,E1 -14285.605,E2 -14285.605} C_VEL
LIN {X 0,Y 340.333,Z 328.555,A -85,B 0,C 180,E1 -14288.736,E2 -14288.736} C_VEL
LIN {X 0,Y 344.496,Z 343.189,A -85,B 0,C 180,E1 -14289.576,E2 -14289.576} C_VEL
LIN {X 0,Y 347.057,Z 354.588,A -85,B 0,C 180,E1 -14290.399,E2 -14290.399} C_VEL
LIN {X 0,Y 347.823,Z 359.769,A -85,B 0,C 180,E1 -14290.819,E2 -14290.819} C_VEL
LIN {X 0,Y 346.728,Z 372.04,A -85,B 0,C 180,E1 -14291.842,E2 -14291.842} C_VEL
LIN {X 0,Y 345.728,Z 381.864,A -85,B 0,C 180,E1 -14292.884,E2 -14292.884} C_VEL
LIN {X 0,Y 344.794,Z 391.681,A -85,B 0,C 180,E1 -14294.179,E2 -14294.179} C_VEL
LIN {X 0,Y 343.739,Z 399.924,A -85,B 0,C 180,E1 -14295.495,E2 -14295.495} C_VEL
LIN {X 0,Y 342.534,Z 408.851,A -85,B 0,C 180,E1 -14297.258,E2 -14297.258} C_VEL
LIN {X 0,Y 341.578,Z 416.016,A -85,B 0,C 180,E1 -14299.029,E2 -14299.029} C_VEL
LIN {X 0,Y 340.701,Z 422.579,A -85,B 0,C 180,E1 -14301.1,E2 -14301.1} C_VEL
LIN {X 0,Y 340.171,Z 426.888,A -85,B 0,C 180,E1 -14302.879,E2 -14302.879} C_VEL
LIN {X 0,Y 339.861,Z 429.158,A -85,B 0,C 180,E1 -14304.065,E2 -14304.065} C_VEL
LIN {X 0,Y 339.636,Z 431.008,A -85,B 0,C 180,E1 -14305.252,E2 -14305.252} C_VEL
LIN {X 0,Y 339.592,Z 432.41,A -85,B 0,C 180,E1 -14306.44,E2 -14306.44} C_VEL
LIN {X 0,Y 339.5,Z 433.398,A -85,B 0,C 180,E1 -14307.627,E2 -14307.627} C_VEL
LIN {X 0,Y 339.346,Z 434.245,A -85,B 0,C 180,E1 -14310,E2 -14310} C_VEL
LIN {X 0,Y 339.498,Z 433.465,A -85,B 0,C 180,E1 -14312.373,E2 -14312.373} C_VEL
LIN {X 0,Y 339.569,Z 432.505,A -85,B 0,C 180,E1 -14313.56,E2 -14313.56} C_VEL
LIN {X 0,Y 339.613,Z 431.155,A -85,B 0,C 180,E1 -14314.748,E2 -14314.748} C_VEL
LIN {X 0,Y 340.037,Z 428.294,A -85,B 0,C 180,E1 -14316.527,E2 -14316.527} C_VEL
LIN {X 0,Y 340.458,Z 424.417,A -85,B 0,C 180,E1 -14318.308,E2 -14318.308} C_VEL
LIN {X 0,Y 341.07,Z 419.391,A -85,B 0,C 180,E1 -14320.087,E2 -14320.087} C_VEL
LIN {X 0,Y 342.002,Z 413.036,A -85,B 0,C 180,E1 -14321.859,E2 -14321.859} C_VEL
LIN {X 0,Y 343.075,Z 405.14,A -85,B 0,C 180,E1 -14323.626,E2 -14323.626} C_VEL
LIN {X 0,Y 344.158,Z 397.064,A -85,B 0,C 180,E1 -14325.092,E2 -14325.092} C_VEL
LIN {X 0,Y 345.291,Z 387.146,A -85,B 0,C 180,E1 -14326.556,E2 -14326.556} C_VEL
LIN {X 0,Y 346.234,Z 377.345,A -85,B 0,C 180,E1 -14327.727,E2 -14327.727} C_VEL
LIN {X 0,Y 347.319,Z 366.694,A -85,B 0,C 180,E1 -14328.737,E2 -14328.737} C_VEL
LIN {X 0,Y 347.763,Z 358.107,A -85,B 0,C 180,E1 -14329.411,E2 -14329.411} C_VEL
LIN {X 0,Y 344.944,Z 345.016,A -85,B 0,C 180,E1 -14330.409,E2 -14330.409} C_VEL
LIN {X 0,Y 341.426,Z 332.409,A -85,B 0,C 180,E1 -14331.168,E2 -14331.168} C_VEL
LIN {X 0,Y 340.361,Z 328.565,A -85,B 0,C 180,E1 -14331.365,E2 -14331.365} C_VEL
LIN {X 0,Y 340.304,Z 322.991,A -85,B 0,C 180,E1 -14334.674,E2 -14334.674} C_VEL
LIN {X 0,Y 340.425,Z 317.125,A -85,B 0,C 180,E1 -14338.348,E2 -14338.348} C_VEL
LIN {X 0,Y 340.645,Z 310.86,A -85,B 0,C 180,E1 -14342.44,E2 -14342.44} C_VEL
LIN {X 0,Y 340.696,Z 307.049,A -85,B 0,C 180,E1 -14345.006,E2 -14345.006} C_VEL
LIN {X 0,Y 340.709,Z 307.047,A -85,B 0,C 180,E1 -14348.385,E2 -14348.385} C_VEL
LIN {X 0,Y 340.701,Z 307.048,A -85,B 0,C 180,E1 -14352.045,E2 -14352.045} C_VEL
LIN {X 0,Y 340.655,Z 307.053,A -85,B 0,C 180,E1 -14353.39,E2 -14353.39} C_VEL
LIN {X 0,Y 339.977,Z 307.14,A -85,B 0,C 180,E1 -14354.376,E2 -14354.376} C_VEL
LIN {X 0,Y 337.114,Z 307.493,A -85,B 0,C 180,E1 -14355.979,E2 -14355.979} C_VEL
LIN {X 0,Y 334.706,Z 307.795,A -85,B 0,C 180,E1 -14357.278,E2 -14357.278} C_VEL
LIN {X 0,Y 333.69,Z 307.919,A -85,B 0,C 180,E1 -14358.283,E2 -14358.283} C_VEL
LIN {X 0,Y 333.616,Z 307.925,A -85,B 0,C 180,E1 -14358.623,E2 -14358.623} C_VEL
LIN {X 0,Y 333.639,Z 307.923,A -85,B 0,C 180,E1 -14362.347,E2 -14362.347} C_VEL
LIN {X 0,Y 333.518,Z 307.935,A -85,B 0,C 180,E1 -14365.322,E2 -14365.322} C_VEL
LIN {X 0,Y 333.417,Z 308.117,A -85,B 0,C 180,E1 -14367.003,E2 -14367.003} C_VEL
LIN {X 0,Y 333.067,Z 315.279,A -85,B 0,C 180,E1 -14371.655,E2 -14371.655} C_VEL
LIN {X 0,Y 332.947,Z 320.676,A -85,B 0,C 180,E1 -14375.185,E2 -14375.185} C_VEL
LIN {X 0,Y 332.847,Z 326.679,A -85,B 0,C 180,E1 -14378.964,E2 -14378.964} C_VEL
LIN {X 0,Y 332.846,Z 329.031,A -85,B 0,C 180,E1 -14380.462,E2 -14380.462} C_VEL
LIN {X 0,Y 335.722,Z 343.873,A -85,B 0,C 180,E1 -14381.295,E2 -14381.295} C_VEL
LIN {X 0,Y 337.803,Z 355.462,A -85,B 0,C 180,E1 -14382.129,E2 -14382.129} C_VEL
LIN {X 0,Y 337.05,Z 368.084,A -85,B 0,C 180,E1 -14383.171,E2 -14383.171} C_VEL
LIN {X 0,Y 336.217,Z 379.719,A -85,B 0,C 180,E1 -14384.387,E2 -14384.387} C_VEL
LIN {X 0,Y 335.432,Z 390.25,A -85,B 0,C 180,E1 -14385.748,E2 -14385.748} C_VEL
LIN {X 0,Y 334.563,Z 399.834,A -85,B 0,C 180,E1 -14387.257,E2 -14387.257} C_VEL
LIN {X 0,Y 333.935,Z 407.807,A -85,B 0,C 180,E1 -14388.774,E2 -14388.774} C_VEL
LIN {X 0,Y 333.295,Z 415.631,A -85,B 0,C 180,E1 -14390.594,E2 -14390.594} C_VEL
LIN {X 0,Y 332.763,Z 422.875,A -85,B 0,C 180,E1 -14392.72,E2 -14392.72} C_VEL
LIN {X 0,Y 332.536,Z 427.641,A -85,B 0,C 180,E1 -14394.543,E2 -14394.543} C_VEL
LIN {X 0,Y 332.373,Z 431.253,A -85,B 0,C 180,E1 -14396.363,E2 -14396.363} C_VEL
LIN {X 0,Y 332.311,Z 433.059,A -85,B 0,C 180,E1 -14397.576,E2 -14397.576} C_VEL
LIN {X 0,Y 332.298,Z 434.445,A -85,B 0,C 180,E1 -14398.788,E2 -14398.788} C_VEL
LIN {X 0,Y 332.31,Z 435.35,A -85,B 0,C 180,E1 -14400,E2 -14400} C_VEL
LIN {X 0,Y 332.367,Z 435.842,A -85,B 0,C 180,E1 -14401.212,E2 -14401.212} C_VEL
LIN {X 0,Y 332.52,Z 435.919,A -85,B 0,C 180,E1 -14402.423,E2 -14402.423} C_VEL
LIN {X 0,Y 332.744,Z 435.516,A -85,B 0,C 180,E1 -14403.633,E2 -14403.633} C_VEL
LIN {X 0,Y 333.002,Z 434.703,A -85,B 0,C 180,E1 -14404.843,E2 -14404.843} C_VEL
LIN {X 0,Y 333.153,Z 433.492,A -85,B 0,C 180,E1 -14406.055,E2 -14406.055} C_VEL
LIN {X 0,Y 333.354,Z 431.805,A -85,B 0,C 180,E1 -14407.267,E2 -14407.267} C_VEL
LIN {X 0,Y 334.249,Z 428.373,A -85,B 0,C 180,E1 -14409.073,E2 -14409.073} C_VEL
LIN {X 0,Y 335.087,Z 423.829,A -85,B 0,C 180,E1 -14410.881,E2 -14410.881} C_VEL
LIN {X 0,Y 336.335,Z 416.954,A -85,B 0,C 180,E1 -14412.981,E2 -14412.981} C_VEL
LIN {X 0,Y 337.745,Z 409.457,A -85,B 0,C 180,E1 -14414.768,E2 -14414.768} C_VEL
LIN {X 0,Y 339.073,Z 401.844,A -85,B 0,C 180,E1 -14416.249,E2 -14416.249} C_VEL
LIN {X 0,Y 340.982,Z 390.656,A -85,B 0,C 180,E1 -14418.009,E2 -14418.009} C_VEL
LIN {X 0,Y 342.457,Z 380.861,A -85,B 0,C 180,E1 -14419.26,E2 -14419.26} C_VEL
LIN {X 0,Y 344.118,Z 368.503,A -85,B 0,C 180,E1 -14420.523,E2 -14420.523} C_VEL
LIN {X 0,Y 344.617,Z 364.175,A -85,B 0,C 180,E1 -14420.906,E2 -14420.906} C_VEL
LIN {X 0,Y 342.314,Z 354.123,A -85,B 0,C 180,E1 -14422.077,E2 -14422.077} C_VEL
LIN {X 0,Y 339.025,Z 344.772,A -85,B 0,C 180,E1 -14423.196,E2 -14423.196} C_VEL
LIN {X 0,Y 335.823,Z 337.495,A -85,B 0,C 180,E1 -14424.084,E2 -14424.084} C_VEL
LIN {X 0,Y 335.146,Z 335.466,A -85,B 0,C 180,E1 -14424.342,E2 -14424.342} C_VEL
LIN {X 0,Y 335.738,Z 329.178,A -85,B 0,C 180,E1 -14428.781,E2 -14428.781} C_VEL
LIN {X 0,Y 336.607,Z 323.457,A -85,B 0,C 180,E1 -14432.878,E2 -14432.878} C_VEL
LIN {X 0,Y 336.544,Z 320.259,A -85,B 0,C 180,E1 -14435.468,E2 -14435.468} C_VEL
LIN {X 0,Y 336.245,Z 318.127,A -85,B 0,C 180,E1 -14437.415,E2 -14437.415} C_VEL
LIN {X 0,Y 335.654,Z 315.251,A -85,B 0,C 180,E1 -14440.473,E2 -14440.473} C_VEL
LIN {X 0,Y 335.246,Z 313.536,A -85,B 0,C 180,E1 -14442.8,E2 -14442.8} C_VEL
LIN {X 0,Y 334.639,Z 313.03,A -85,B 0,C 180,E1 -14444.377,E2 -14444.377} C_VEL
LIN {X 0,Y 335.917,Z 319.76,A -85,B 0,C 180,E1 -14447.971,E2 -14447.971} C_VEL
LIN {X 0,Y 337.204,Z 326.276,A -85,B 0,C 180,E1 -14451.299,E2 -14451.299} C_VEL
LIN {X 0,Y 337.524,Z 329.47,A -85,B 0,C 180,E1 -14452.854,E2 -14452.854} C_VEL
LIN {X 0,Y 336.76,Z 335.65,A -85,B 0,C 180,E1 -14455.703,E2 -14455.703} C_VEL
LIN {X 0,Y 335.8,Z 343.195,A -85,B 0,C 180,E1 -14459.103,E2 -14459.103} C_VEL
LIN {X 0,Y 334.771,Z 352.414,A -85,B 0,C 180,E1 -14463.169,E2 -14463.169} C_VEL
LIN {X 0,Y 334.084,Z 359.564,A -85,B 0,C 180,E1 -14466.276,E2 -14466.276} C_VEL
LIN {X 0,Y 334.814,Z 363.441,A -85,B 0,C 180,E1 -14466.575,E2 -14466.575} C_VEL
LIN {X 0,Y 337.862,Z 376.511,A -85,B 0,C 180,E1 -14467.659,E2 -14467.659} C_VEL
LIN {X 0,Y 338.903,Z 384.861,A -85,B 0,C 180,E1 -14468.347,E2 -14468.347} C_VEL
LIN {X 0,Y 339.54,Z 397.951,A -85,B 0,C 180,E1 -14469.504,E2 -14469.504} C_VEL
LIN {X 0,Y 339.811,Z 410.409,A -85,B 0,C 180,E1 -14470.833,E2 -14470.833} C_VEL
LIN {X 0,Y 338.133,Z 421.811,A -85,B 0,C 180,E1 -14472.147,E2 -14472.147} C_VEL
LIN {X 0,Y 336.447,Z 433.346,A -85,B 0,C 180,E1 -14473.831,E2 -14473.831} C_VEL
LIN {X 0,Y 335.22,Z 442.257,A -85,B 0,C 180,E1 -14475.429,E2 -14475.429} C_VEL
LIN {X 0,Y 334.055,Z 450.484,A -85,B 0,C 180,E1 -14477.238,E2 -14477.238} C_VEL
LIN {X 0,Y 333.231,Z 457.219,A -85,B 0,C 180,E1 -14479.058,E2 -14479.058} C_VEL
LIN {X 0,Y 332.646,Z 462.662,A -85,B 0,C 180,E1 -14480.883,E2 -14480.883} C_VEL
LIN {X 0,Y 332.362,Z 466.946,A -85,B 0,C 180,E1 -14482.711,E2 -14482.711} C_VEL
LIN {X 0,Y 332.221,Z 469.192,A -85,B 0,C 180,E1 -14483.928,E2 -14483.928} C_VEL
LIN {X 0,Y 332.143,Z 470.983,A -85,B 0,C 180,E1 -14485.145,E2 -14485.145} C_VEL
LIN {X 0,Y 332.136,Z 472.363,A -85,B 0,C 180,E1 -14486.36,E2 -14486.36} C_VEL
LIN {X 0,Y 332.114,Z 473.295,A -85,B 0,C 180,E1 -14487.574,E2 -14487.574} C_VEL
LIN {X 0,Y 332.293,Z 473.79,A -85,B 0,C 180,E1 -14488.788,E2 -14488.788} C_VEL
LIN {X 0,Y 332.338,Z 473.867,A -85,B 0,C 180,E1 -14490,E2 -14490} C_VEL
LIN {X 0,Y 332.33,Z 473.517,A -85,B 0,C 180,E1 -14491.212,E2 -14491.212} C_VEL
LIN {X 0,Y 332.133,Z 471.683,A -85,B 0,C 180,E1 -14493.64,E2 -14493.64} C_VEL
LIN {X 0,Y 332.181,Z 470.232,A -85,B 0,C 180,E1 -14494.855,E2 -14494.855} C_VEL
LIN {X 0,Y 332.279,Z 467.215,A -85,B 0,C 180,E1 -14496.68,E2 -14496.68} C_VEL
LIN {X 0,Y 332.506,Z 463.121,A -85,B 0,C 180,E1 -14498.508,E2 -14498.508} C_VEL
LIN {X 0,Y 333.079,Z 456.819,A -85,B 0,C 180,E1 -14500.639,E2 -14500.639} C_VEL
LIN {X 0,Y 334.021,Z 448.795,A -85,B 0,C 180,E1 -14502.764,E2 -14502.764} C_VEL
LIN {X 0,Y 335.11,Z 440.746,A -85,B 0,C 180,E1 -14504.576,E2 -14504.576} C_VEL
LIN {X 0,Y 336.47,Z 431.017,A -85,B 0,C 180,E1 -14506.378,E2 -14506.378} C_VEL
LIN {X 0,Y 338.213,Z 420.163,A -85,B 0,C 180,E1 -14508.005,E2 -14508.005} C_VEL
LIN {X 0,Y 339.861,Z 409.419,A -85,B 0,C 180,E1 -14509.321,E2 -14509.321} C_VEL
LIN {X 0,Y 339.763,Z 398.248,A -85,B 0,C 180,E1 -14510.588,E2 -14510.588} C_VEL
LIN {X 0,Y 339.486,Z 386.133,A -85,B 0,C 180,E1 -14511.76,E2 -14511.76} C_VEL
LIN {X 0,Y 338.087,Z 374.984,A -85,B 0,C 180,E1 -14512.777,E2 -14512.777} C_VEL
LIN {X 0,Y 335.215,Z 361.868,A -85,B 0,C 180,E1 -14513.946,E2 -14513.946} C_VEL
LIN {X 0,Y 334.195,Z 358.198,A -85,B 0,C 180,E1 -14514.272,E2 -14514.272} C_VEL
LIN {X 0,Y 334.166,Z 357.508,A -85,B 0,C 180,E1 -14514.377,E2 -14514.377} C_VEL
LIN {X 0,Y 335.064,Z 349.159,A -85,B 0,C 180,E1 -14518.242,E2 -14518.242} C_VEL
LIN {X 0,Y 336.279,Z 341.213,A -85,B 0,C 180,E1 -14522.204,E2 -14522.204} C_VEL
LIN {X 0,Y 337.812,Z 333.711,A -85,B 0,C 180,E1 -14526.365,E2 -14526.365} C_VEL
LIN {X 0,Y 338.086,Z 331.399,A -85,B 0,C 180,E1 -14527.821,E2 -14527.821} C_VEL
LIN {X 0,Y 337.604,Z 328.187,A -85,B 0,C 180,E1 -14530.191,E2 -14530.191} C_VEL
LIN {X 0,Y 336.889,Z 324.482,A -85,B 0,C 180,E1 -14533.506,E2 -14533.506} C_VEL
LIN {X 0,Y 336.333,Z 321.481,A -85,B 0,C 180,E1 -14537.001,E2 -14537.001} C_VEL
LIN {X 0,Y 336.04,Z 319.87,A -85,B 0,C 180,E1 -14539.583,E2 -14539.583} C_VEL
LIN {X 0,Y 335.781,Z 318.572,A -85,B 0,C 180,E1 -14542.689,E2 -14542.689} C_VEL
LIN {X 0,Y 335.587,Z 317.96,A -85,B 0,C 180,E1 -14545.567,E2 -14545.567} C_VEL
LIN {X 0,Y 335.492,Z 317.86,A -85,B 0,C 180,E1 -14549.192,E2 -14549.192} C_VEL
LIN {X 0,Y 335.518,Z 318.336,A -85,B 0,C 180,E1 -14552.559,E2 -14552.559} C_VEL
LIN {X 0,Y 335.451,Z 319.362,A -85,B 0,C 180,E1 -14555.788,E2 -14555.788} C_VEL
LIN {X 0,Y 335.942,Z 320.808,A -85,B 0,C 180,E1 -14555.955,E2 -14555.955} C_VEL
LIN {X 0,Y 341.415,Z 331.101,A -85,B 0,C 180,E1 -14557.475,E2 -14557.475} C_VEL
LIN {X 0,Y 344.786,Z 339.969,A -85,B 0,C 180,E1 -14558.671,E2 -14558.671} C_VEL
LIN {X 0,Y 345.796,Z 343.622,A -85,B 0,C 180,E1 -14559.146,E2 -14559.146} C_VEL
LIN {X 0,Y 344.075,Z 357.014,A -85,B 0,C 180,E1 -14560.469,E2 -14560.469} C_VEL
LIN {X 0,Y 342.537,Z 367.461,A -85,B 0,C 180,E1 -14561.766,E2 -14561.766} C_VEL
LIN {X 0,Y 340.919,Z 377.048,A -85,B 0,C 180,E1 -14563.225,E2 -14563.225} C_VEL
LIN {X 0,Y 339.455,Z 385.033,A -85,B 0,C 180,E1 -14564.694,E2 -14564.694} C_VEL
LIN {X 0,Y 338.009,Z 392.847,A -85,B 0,C 180,E1 -14566.472,E2 -14566.472} C_VEL
LIN {X 0,Y 336.817,Z 398.206,A -85,B 0,C 180,E1 -14567.956,E2 -14567.956} C_VEL
LIN {X 0,Y 335.835,Z 403.211,A -85,B 0,C 180,E1 -14569.693,E2 -14569.693} C_VEL
LIN {X 0,Y 334.781,Z 407.391,A -85,B 0,C 180,E1 -14571.55,E2 -14571.55} C_VEL
LIN {X 0,Y 334.347,Z 409.447,A -85,B 0,C 180,E1 -14572.755,E2 -14572.755} C_VEL
LIN {X 0,Y 333.957,Z 411.067,A -85,B 0,C 180,E1 -14573.96,E2 -14573.96} C_VEL
LIN {X 0,Y 333.564,Z 412.215,A -85,B 0,C 180,E1 -14575.166,E2 -14575.166} C_VEL
LIN {X 0,Y 333.169,Z 412.969,A -85,B 0,C 180,E1 -14576.372,E2 -14576.372} C_VEL
LIN {X 0,Y 332.876,Z 413.314,A -85,B 0,C 180,E1 -14577.58,E2 -14577.58} C_VEL
LIN {X 0,Y 332.713,Z 413.195,A -85,B 0,C 180,E1 -14578.79,E2 -14578.79} C_VEL
LIN {X 0,Y 332.655,Z 412.644,A -85,B 0,C 180,E1 -14580,E2 -14580} C_VEL
LIN {X 0,Y 332.693,Z 411.68,A -85,B 0,C 180,E1 -14581.211,E2 -14581.211} C_VEL
LIN {X 0,Y 332.715,Z 410.293,A -85,B 0,C 180,E1 -14582.421,E2 -14582.421} C_VEL
LIN {X 0,Y 332.993,Z 407.36,A -85,B 0,C 180,E1 -14584.236,E2 -14584.236} C_VEL
LIN {X 0,Y 333.119,Z 403.37,A -85,B 0,C 180,E1 -14586.055,E2 -14586.055} C_VEL
LIN {X 0,Y 333.475,Z 397.346,A -85,B 0,C 180,E1 -14588.134,E2 -14588.134} C_VEL
LIN {X 0,Y 333.965,Z 390.493,A -85,B 0,C 180,E1 -14589.998,E2 -14589.998} C_VEL
LIN {X 0,Y 334.669,Z 382.146,A -85,B 0,C 180,E1 -14591.815,E2 -14591.815} C_VEL
LIN {X 0,Y 335.528,Z 371.839,A -85,B 0,C 180,E1 -14593.63,E2 -14593.63} C_VEL
LIN {X 0,Y 336.43,Z 361.162,A -85,B 0,C 180,E1 -14595.137,E2 -14595.137} C_VEL
LIN {X 0,Y 337.163,Z 349.396,A -85,B 0,C 180,E1 -14596.494,E2 -14596.494} C_VEL
LIN {X 0,Y 338.013,Z 335.958,A -85,B 0,C 180,E1 -14597.703,E2 -14597.703} C_VEL
LIN {X 0,Y 338.221,Z 329.872,A -85,B 0,C 180,E1 -14598.161,E2 -14598.161} C_VEL
LIN {X 0,Y 335.195,Z 316.275,A -85,B 0,C 180,E1 -14599.111,E2 -14599.111} C_VEL
LIN {X 0,Y 333.128,Z 307.991,A -85,B 0,C 180,E1 -14599.6,E2 -14599.6} C_VEL
LIN {X 0,Y 333.367,Z 307.956,A -85,B 0,C 180,E1 -14602.301,E2 -14602.301} C_VEL
LIN {X 0,Y 333.609,Z 307.926,A -85,B 0,C 180,E1 -14605.06,E2 -14605.06} C_VEL
LIN {X 0,Y 333.673,Z 307.917,A -85,B 0,C 180,E1 -14607.794,E2 -14607.794} C_VEL
LIN {X 0,Y 333.692,Z 307.915,A -85,B 0,C 180,E1 -14610.363,E2 -14610.363} C_VEL
LIN {X 0,Y 333.676,Z 307.916,A -85,B 0,C 180,E1 -14614.659,E2 -14614.659} C_VEL
LIN {X 0,Y 333.654,Z 307.927,A -85,B 0,C 180,E1 -14617.651,E2 -14617.651} C_VEL
LIN {X 0,Y 333.649,Z 307.927,A -85,B 0,C 180,E1 -14620.767,E2 -14620.767} C_VEL
LIN {X 0,Y 333.596,Z 307.931,A -85,B 0,C 180,E1 -14624.251,E2 -14624.251} C_VEL
LIN {X 0,Y 333.644,Z 307.926,A -85,B 0,C 180,E1 -14627.619,E2 -14627.619} C_VEL
LIN {X 0,Y 333.653,Z 307.926,A -85,B 0,C 180,E1 -14631.202,E2 -14631.202} C_VEL
LIN {X 0,Y 333.663,Z 308.052,A -85,B 0,C 180,E1 -14634.972,E2 -14634.972} C_VEL
LIN {X 0,Y 333.742,Z 310.749,A -85,B 0,C 180,E1 -14636.803,E2 -14636.803} C_VEL
LIN {X 0,Y 333.455,Z 317.148,A -85,B 0,C 180,E1 -14641.003,E2 -14641.003} C_VEL
LIN {X 0,Y 333.331,Z 323.541,A -85,B 0,C 180,E1 -14645.059,E2 -14645.059} C_VEL
LIN {X 0,Y 333.355,Z 328.929,A -85,B 0,C 180,E1 -14648.278,E2 -14648.278} C_VEL
LIN {X 0,Y 337.45,Z 343.228,A -85,B 0,C 180,E1 -14649.113,E2 -14649.113} C_VEL
LIN {X 0,Y 340.18,Z 355.177,A -85,B 0,C 180,E1 -14649.999,E2 -14649.999} C_VEL
LIN {X 0,Y 341.098,Z 360.383,A -85,B 0,C 180,E1 -14650.443,E2 -14650.443} C_VEL
LIN {X 0,Y 340.011,Z 372.443,A -85,B 0,C 180,E1 -14651.47,E2 -14651.47} C_VEL
LIN {X 0,Y 338.926,Z 382.602,A -85,B 0,C 180,E1 -14652.571,E2 -14652.571} C_VEL
LIN {X 0,Y 337.866,Z 393.088,A -85,B 0,C 180,E1 -14654.001,E2 -14654.001} C_VEL
LIN {X 0,Y 336.591,Z 401.952,A -85,B 0,C 180,E1 -14655.489,E2 -14655.489} C_VEL
LIN {X 0,Y 335.458,Z 410.582,A -85,B 0,C 180,E1 -14657.292,E2 -14657.292} C_VEL
LIN {X 0,Y 334.442,Z 417.5,A -85,B 0,C 180,E1 -14659.098,E2 -14659.098} C_VEL
LIN {X 0,Y 333.691,Z 422.994,A -85,B 0,C 180,E1 -14660.911,E2 -14660.911} C_VEL
LIN {X 0,Y 333.131,Z 427.303,A -85,B 0,C 180,E1 -14662.728,E2 -14662.728} C_VEL
LIN {X 0,Y 332.834,Z 429.572,A -85,B 0,C 180,E1 -14663.939,E2 -14663.939} C_VEL
LIN {X 0,Y 332.574,Z 431.423,A -85,B 0,C 180,E1 -14665.151,E2 -14665.151} C_VEL
LIN {X 0,Y 332.509,Z 432.826,A -85,B 0,C 180,E1 -14666.364,E2 -14666.364} C_VEL
LIN {X 0,Y 332.429,Z 433.812,A -85,B 0,C 180,E1 -14667.577,E2 -14667.577} C_VEL
LIN {X 0,Y 332.286,Z 434.658,A -85,B 0,C 180,E1 -14670,E2 -14670} C_VEL
LIN {X 0,Y 332.426,Z 433.879,A -85,B 0,C 180,E1 -14672.423,E2 -14672.423} C_VEL
LIN {X 0,Y 332.486,Z 432.92,A -85,B 0,C 180,E1 -14673.636,E2 -14673.636} C_VEL
LIN {X 0,Y 332.553,Z 431.568,A -85,B 0,C 180,E1 -14674.849,E2 -14674.849} C_VEL
LIN {X 0,Y 333.009,Z 428.706,A -85,B 0,C 180,E1 -14676.666,E2 -14676.666} C_VEL
LIN {X 0,Y 333.447,Z 424.829,A -85,B 0,C 180,E1 -14678.484,E2 -14678.484} C_VEL
LIN {X 0,Y 334.107,Z 419.801,A -85,B 0,C 180,E1 -14680.3,E2 -14680.3} C_VEL
LIN {X 0,Y 335.052,Z 413.447,A -85,B 0,C 180,E1 -14682.108,E2 -14682.108} C_VEL
LIN {X 0,Y 336.187,Z 405.547,A -85,B 0,C 180,E1 -14683.911,E2 -14683.911} C_VEL
LIN {X 0,Y 337.31,Z 397.469,A -85,B 0,C 180,E1 -14685.406,E2 -14685.406} C_VEL
LIN {X 0,Y 338.501,Z 387.546,A -85,B 0,C 180,E1 -14686.898,E2 -14686.898} C_VEL
LIN {X 0,Y 339.507,Z 377.739,A -85,B 0,C 180,E1 -14688.09,E2 -14688.09} C_VEL
LIN {X 0,Y 340.632,Z 367.081,A -85,B 0,C 180,E1 -14689.119,E2 -14689.119} C_VEL
LIN {X 0,Y 341.121,Z 360.074,A -85,B 0,C 180,E1 -14689.687,E2 -14689.687} C_VEL
LIN {X 0,Y 338.576,Z 347.708,A -85,B 0,C 180,E1 -14690.68,E2 -14690.68} C_VEL
LIN {X 0,Y 335.048,Z 334.65,A -85,B 0,C 180,E1 -14691.526,E2 -14691.526} C_VEL
LIN {X 0,Y 333.374,Z 328.928,A -85,B 0,C 180,E1 -14691.839,E2 -14691.839} C_VEL
LIN {X 0,Y 333.345,Z 322.651,A -85,B 0,C 180,E1 -14695.607,E2 -14695.607} C_VEL
LIN {X 0,Y 333.452,Z 317.32,A -85,B 0,C 180,E1 -14698.997,E2 -14698.997} C_VEL
LIN {X 0,Y 333.77,Z 310.922,A -85,B 0,C 180,E1 -14703.194,E2 -14703.194} C_VEL
LIN {X 0,Y 333.649,Z 307.927,A -85,B 0,C 180,E1 -14705.314,E2 -14705.314} C_VEL
LIN {X 0,Y 333.648,Z 307.926,A -85,B 0,C 180,E1 -14709.192,E2 -14709.192} C_VEL
LIN {X 0,Y 333.635,Z 307.931,A -85,B 0,C 180,E1 -14712.5,E2 -14712.5} C_VEL
LIN {X 0,Y 333.599,Z 307.931,A -85,B 0,C 180,E1 -14715.955,E2 -14715.955} C_VEL
LIN {X 0,Y 333.616,Z 307.925,A -85,B 0,C 180,E1 -14718.623,E2 -14718.623} C_VEL
LIN {X 0,Y 332.97,Z 308.01,A -85,B 0,C 180,E1 -14719.63,E2 -14719.63} C_VEL
LIN {X 0,Y 330.116,Z 308.362,A -85,B 0,C 180,E1 -14721.269,E2 -14721.269} C_VEL
LIN {X 0,Y 327.677,Z 308.667,A -85,B 0,C 180,E1 -14722.596,E2 -14722.596} C_VEL
LIN {X 0,Y 326.619,Z 308.801,A -85,B 0,C 180,E1 -14723.623,E2 -14723.623} C_VEL
LIN {X 0,Y 326.528,Z 308.807,A -85,B 0,C 180,E1 -14723.972,E2 -14723.972} C_VEL
LIN {X 0,Y 326.39,Z 308.916,A -85,B 0,C 180,E1 -14726.923,E2 -14726.923} C_VEL
LIN {X 0,Y 326.05,Z 315.135,A -85,B 0,C 180,E1 -14730.988,E2 -14730.988} C_VEL
LIN {X 0,Y 325.907,Z 321.131,A -85,B 0,C 180,E1 -14734.919,E2 -14734.919} C_VEL
LIN {X 0,Y 325.812,Z 326.694,A -85,B 0,C 180,E1 -14738.487,E2 -14738.487} C_VEL
LIN {X 0,Y 325.771,Z 329.432,A -85,B 0,C 180,E1 -14740.219,E2 -14740.219} C_VEL
LIN {X 0,Y 328.446,Z 343.389,A -85,B 0,C 180,E1 -14741,E2 -14741} C_VEL
LIN {X 0,Y 330.742,Z 355.559,A -85,B 0,C 180,E1 -14741.894,E2 -14741.894} C_VEL
LIN {X 0,Y 330.033,Z 368.702,A -85,B 0,C 180,E1 -14743.006,E2 -14743.006} C_VEL
LIN {X 0,Y 329.215,Z 379.939,A -85,B 0,C 180,E1 -14744.206,E2 -14744.206} C_VEL
LIN {X 0,Y 328.407,Z 390.521,A -85,B 0,C 180,E1 -14745.595,E2 -14745.595} C_VEL
LIN {X 0,Y 327.453,Z 401.026,A -85,B 0,C 180,E1 -14747.291,E2 -14747.291} C_VEL
LIN {X 0,Y 326.675,Z 410.261,A -85,B 0,C 180,E1 -14749.15,E2 -14749.15} C_VEL
LIN {X 0,Y 326.093,Z 417.74,A -85,B 0,C 180,E1 -14751.01,E2 -14751.01} C_VEL
LIN {X 0,Y 325.709,Z 422.794,A -85,B 0,C 180,E1 -14752.561,E2 -14752.561} C_VEL
LIN {X 0,Y 325.462,Z 427.703,A -85,B 0,C 180,E1 -14754.424,E2 -14754.424} C_VEL
LIN {X 0,Y 325.292,Z 431.429,A -85,B 0,C 180,E1 -14756.284,E2 -14756.284} C_VEL
LIN {X 0,Y 325.218,Z 433.294,A -85,B 0,C 180,E1 -14757.523,E2 -14757.523} C_VEL
LIN {X 0,Y 325.205,Z 434.745,A -85,B 0,C 180,E1 -14758.762,E2 -14758.762} C_VEL
LIN {X 0,Y 325.25,Z 435.744,A -85,B 0,C 180,E1 -14760,E2 -14760} C_VEL
LIN {X 0,Y 325.31,Z 436.289,A -85,B 0,C 180,E1 -14761.238,E2 -14761.238} C_VEL
LIN {X 0,Y 325.47,Z 436.422,A -85,B 0,C 180,E1 -14762.475,E2 -14762.475} C_VEL
LIN {X 0,Y 325.706,Z 436.115,A -85,B 0,C 180,E1 -14763.711,E2 -14763.711} C_VEL
LIN {X 0,Y 325.974,Z 435.36,A -85,B 0,C 180,E1 -14764.947,E2 -14764.947} C_VEL
LIN {X 0,Y 326.135,Z 434.217,A -85,B 0,C 180,E1 -14766.185,E2 -14766.185} C_VEL
LIN {X 0,Y 326.359,Z 432.622,A -85,B 0,C 180,E1 -14767.424,E2 -14767.424} C_VEL
LIN {X 0,Y 327.31,Z 429.286,A -85,B 0,C 180,E1 -14769.267,E2 -14769.267} C_VEL
LIN {X 0,Y 328.196,Z 424.895,A -85,B 0,C 180,E1 -14771.112,E2 -14771.112} C_VEL
LIN {X 0,Y 329.549,Z 418.225,A -85,B 0,C 180,E1 -14773.253,E2 -14773.253} C_VEL
LIN {X 0,Y 331.035,Z 410.873,A -85,B 0,C 180,E1 -14775.074,E2 -14775.074} C_VEL
LIN {X 0,Y 332.448,Z 403.512,A -85,B 0,C 180,E1 -14776.582,E2 -14776.582} C_VEL
LIN {X 0,Y 334.163,Z 394.645,A -85,B 0,C 180,E1 -14778.072,E2 -14778.072} C_VEL
LIN {X 0,Y 335.899,Z 383.876,A -85,B 0,C 180,E1 -14779.558,E2 -14779.558} C_VEL
LIN {X 0,Y 337.507,Z 373.461,A -85,B 0,C 180,E1 -14780.732,E2 -14780.732} C_VEL
LIN {X 0,Y 338.461,Z 366.102,A -85,B 0,C 180,E1 -14781.43,E2 -14781.43} C_VEL
LIN {X 0,Y 336.225,Z 356.107,A -85,B 0,C 180,E1 -14782.668,E2 -14782.668} C_VEL
LIN {X 0,Y 331.515,Z 343.182,A -85,B 0,C 180,E1 -14784.343,E2 -14784.343} C_VEL
LIN {X 0,Y 328.442,Z 336.226,A -85,B 0,C 180,E1 -14785.299,E2 -14785.299} C_VEL
LIN {X 0,Y 329.096,Z 330.587,A -85,B 0,C 180,E1 -14789.418,E2 -14789.418} C_VEL
LIN {X 0,Y 329.734,Z 326.889,A -85,B 0,C 180,E1 -14792.199,E2 -14792.199} C_VEL
LIN {X 0,Y 330.004,Z 324.783,A -85,B 0,C 180,E1 -14793.842,E2 -14793.842} C_VEL
LIN {X 0,Y 329.787,Z 321.75,A -85,B 0,C 180,E1 -14796.634,E2 -14796.634} C_VEL
LIN {X 0,Y 329.344,Z 318.841,A -85,B 0,C 180,E1 -14799.806,E2 -14799.806} C_VEL
LIN {X 0,Y 329.084,Z 317.502,A -85,B 0,C 180,E1 -14801.628,E2 -14801.628} C_VEL
LIN {X 0,Y 328.669,Z 316.602,A -85,B 0,C 180,E1 -14803.362,E2 -14803.362} C_VEL
LIN {X 0,Y 327.977,Z 316.141,A -85,B 0,C 180,E1 -14805.317,E2 -14805.317} C_VEL
LIN {X 0,Y 329.486,Z 323.763,A -85,B 0,C 180,E1 -14809.403,E2 -14809.403} C_VEL
LIN {X 0,Y 330.392,Z 328.656,A -85,B 0,C 180,E1 -14811.911,E2 -14811.911} C_VEL
LIN {X 0,Y 330.399,Z 331.8,A -85,B 0,C 180,E1 -14813.445,E2 -14813.445} C_VEL
LIN {X 0,Y 329.313,Z 339.488,A -85,B 0,C 180,E1 -14817.029,E2 -14817.029} C_VEL
LIN {X 0,Y 328.314,Z 347.101,A -85,B 0,C 180,E1 -14820.505,E2 -14820.505} C_VEL
LIN {X 0,Y 327.418,Z 355.684,A -85,B 0,C 180,E1 -14824.36,E2 -14824.36} C_VEL
LIN {X 0,Y 327.221,Z 357.732,A -85,B 0,C 180,E1 -14825.24,E2 -14825.24} C_VEL
LIN {X 0,Y 327.976,Z 361.65,A -85,B 0,C 180,E1 -14825.571,E2 -14825.571} C_VEL
LIN {X 0,Y 328.83,Z 364.756,A -85,B 0,C 180,E1 -14825.861,E2 -14825.861} C_VEL
LIN {X 0,Y 331.518,Z 376.74,A -85,B 0,C 180,E1 -14826.934,E2 -14826.934} C_VEL
LIN {X 0,Y 332.665,Z 384.548,A -85,B 0,C 180,E1 -14827.649,E2 -14827.649} C_VEL
LIN {X 0,Y 333.129,Z 397.392,A -85,B 0,C 180,E1 -14828.83,E2 -14828.83} C_VEL
LIN {X 0,Y 333.355,Z 409.133,A -85,B 0,C 180,E1 -14830.126,E2 -14830.126} C_VEL
LIN {X 0,Y 332.611,Z 415.699,A -85,B 0,C 180,E1 -14830.882,E2 -14830.882} C_VEL
LIN {X 0,Y 330.968,Z 425.946,A -85,B 0,C 180,E1 -14832.227,E2 -14832.227} C_VEL
LIN {X 0,Y 329.317,Z 436.239,A -85,B 0,C 180,E1 -14833.893,E2 -14833.893} C_VEL
LIN {X 0,Y 327.924,Z 445.481,A -85,B 0,C 180,E1 -14835.731,E2 -14835.731} C_VEL
LIN {X 0,Y 326.592,Z 454.133,A -85,B 0,C 180,E1 -14837.889,E2 -14837.889} C_VEL
LIN {X 0,Y 325.803,Z 460.928,A -85,B 0,C 180,E1 -14840.063,E2 -14840.063} C_VEL
LIN {X 0,Y 325.354,Z 465.48,A -85,B 0,C 180,E1 -14841.929,E2 -14841.929} C_VEL
LIN {X 0,Y 325.131,Z 469.114,A -85,B 0,C 180,E1 -14843.899,E2 -14843.899} C_VEL
LIN {X 0,Y 325.058,Z 472.052,A -85,B 0,C 180,E1 -14846.281,E2 -14846.281} C_VEL
LIN {X 0,Y 325.024,Z 472.92,A -85,B 0,C 180,E1 -14847.521,E2 -14847.521} C_VEL
LIN {X 0,Y 325.194,Z 473.385,A -85,B 0,C 180,E1 -14848.762,E2 -14848.762} C_VEL
LIN {X 0,Y 325.276,Z 473.435,A -85,B 0,C 180,E1 -14850,E2 -14850} C_VEL
LIN {X 0,Y 325.263,Z 473.022,A -85,B 0,C 180,E1 -14851.238,E2 -14851.238} C_VEL
LIN {X 0,Y 325.058,Z 471.267,A -85,B 0,C 180,E1 -14853.719,E2 -14853.719} C_VEL
LIN {X 0,Y 325.104,Z 469.816,A -85,B 0,C 180,E1 -14854.961,E2 -14854.961} C_VEL
LIN {X 0,Y 325.202,Z 466.797,A -85,B 0,C 180,E1 -14856.826,E2 -14856.826} C_VEL
LIN {X 0,Y 325.44,Z 462.703,A -85,B 0,C 180,E1 -14858.695,E2 -14858.695} C_VEL
LIN {X 0,Y 326.055,Z 456.402,A -85,B 0,C 180,E1 -14860.871,E2 -14860.871} C_VEL
LIN {X 0,Y 327.458,Z 446.175,A -85,B 0,C 180,E1 -14863.656,E2 -14863.656} C_VEL
LIN {X 0,Y 328.592,Z 438.487,A -85,B 0,C 180,E1 -14865.362,E2 -14865.362} C_VEL
LIN {X 0,Y 329.98,Z 429.503,A -85,B 0,C 180,E1 -14867.029,E2 -14867.029} C_VEL
LIN {X 0,Y 331.881,Z 418.545,A -85,B 0,C 180,E1 -14868.681,E2 -14868.681} C_VEL
LIN {X 0,Y 333.216,Z 410.366,A -85,B 0,C 180,E1 -14869.722,E2 -14869.722} C_VEL
LIN {X 0,Y 333.311,Z 397.838,A -85,B 0,C 180,E1 -14871.205,E2 -14871.205} C_VEL
LIN {X 0,Y 333.139,Z 386.937,A -85,B 0,C 180,E1 -14872.317,E2 -14872.317} C_VEL
LIN {X 0,Y 331.84,Z 376.053,A -85,B 0,C 180,E1 -14873.388,E2 -14873.388} C_VEL
LIN {X 0,Y 329.404,Z 364.621,A -85,B 0,C 180,E1 -14874.51,E2 -14874.51} C_VEL
LIN {X 0,Y 327.32,Z 356.429,A -85,B 0,C 180,E1 -14875.333,E2 -14875.333} C_VEL
